(* IEC 61131-3 sources: Supremica/examples/ilprograms, 2 files *)

(* ---- ballProcess.il ---- *)
JAVA_BLOCK OnDelayTimer
	VAR_IN_OUT
		tonIN : BOOL;
		tonPT : DINT;
		tonET : DINT;
		tonQ  : BOOL;
	END_VAR
END_JAVA_BLOCK
FUNCTION_BLOCK TON
	VAR_IN_OUT
		tonIN : BOOL;
		tonPT : DINT;
		tonET : DINT;
		tonQ  : BOOL;
	END_VAR
	VAR
		odt : OnDelayTimer;
	END_VAR
	LD  tonIN
	ST  odt.tonIN
	LD  tonPT
	ST  odt.tonPT
	CAL odt
	LD  odt.tonET
	ST  tonET
	LD  odt.tonQ
	ST  tonQ
END_FUNCTION_BLOCK
(* This file is automatically generated from Supremica *)
(* Supremica version: 200206130257 *)
(* This file was generated at: Jun 13, 2002 6:24:47 AM *)
PROGRAM AutomaticallyGeneratedProgram
	VAR (* Internal variables *)
		si_6 AT %IX6 : BOOL; (* LitenKula *)
		si_2 AT %IX2 : BOOL; (* KulaMatlyft *)
		si_22 AT %IX22 : BOOL; (* KulaFast *)
		si_24 AT %IX24 : BOOL; (* ManuellStart *)
		si_16 AT %IX16 : BOOL; (* PlockaVan2 *)
		si_0 AT %IX0 : BOOL; (* KulaPortvakt *)
		si_13 AT %IX13 : BOOL; (* PlockaVan1 *)
		si_23 AT %IX23 : BOOL; (* Autostart *)
		si_4 AT %IX4 : BOOL; (* KulaMatstation *)
		si_14 AT %IX14 : BOOL; (* HissVan2 *)
		si_11 AT %IX11 : BOOL; (* HissVan1 *)
		si_15 AT %IX15 : BOOL; (* KulaVan2 *)
		si_12 AT %IX12 : BOOL; (* KulaVan1 *)
		si_25 AT %IX25 : BOOL; (* NodStopp *)
		si_21 AT %IX21 : BOOL; (* ArmVan2 *)
		si_3 AT %IX3 : BOOL; (* MatlyftUppe *)
		si_7 AT %IX7 : BOOL; (* HissNere *)
		si_20 AT %IX20 : BOOL; (* ArmVan1 *)
		si_17 AT %IX17 : BOOL; (* ArmHemma *)
		si_26 AT %IX26 : BOOL; (* LarmKvittering *)
		si_1 AT %IX1 : BOOL; (* MatlyftNere *)
		si_5 AT %IX5 : BOOL; (* StorKula *)
		si_10 AT %IX10 : BOOL; (* KulaHiss *)
		so_11 AT %QX11 : BOOL; (* UtVan2 *)
		so_7 AT %QX7 : BOOL; (* UtVan1 *)
		so_12 AT %QX12 : BOOL; (* LyftVan2 *)
		so_0 AT %QX0 : BOOL; (* InPortvakt *)
		so_10 AT %QX10 : BOOL; (* LyftVan1 *)
		so_15 AT %QX15 : BOOL; (* VridArmHoger *)
		so_3 AT %QX3 : BOOL; (* UrMatning *)
		so_14 AT %QX14 : BOOL; (* UppArmVan2 *)
		so_2 AT %QX2 : BOOL; (* UppMatlyft *)
		so_16 AT %QX16 : BOOL; (* Sug *)
		so_13 AT %QX13 : BOOL; (* UppArmVan1 *)
		so_6 AT %QX6 : BOOL; (* UppHissVan2 *)
		so_5 AT %QX5 : BOOL; (* UppHissVan1 *)
		so_1 AT %QX1 : BOOL; (* UrPortvakt *)
		so_4 AT %QX4 : BOOL; (* Mat *)
	END_VAR

	VAR (* Internal variables *)
		e_0 : BOOL; (* arm.allocate_lower_buffer controllable *)
		e_1 : BOOL; (* arm.allocate_upper_buffer controllable *)
		e_2 : BOOL; (* arm.lower_lower_buffer controllable *)
		e_3 : BOOL; (* arm.lower_upper_buffer controllable *)
		e_4 : BOOL; (* arm.raise_lower_buffer controllable *)
		e_5 : BOOL; (* arm.raise_upper_buffer controllable *)
		e_6 : BOOL; (* arm.release_lower_buffer controllable *)
		e_7 : BOOL; (* arm.release_upper_buffer controllable *)
		e_8 : BOOL; (* button.automatic.pressed uncontrollable *)
		e_9 : BOOL; (* button.automatic.released uncontrollable *)
		e_10 : BOOL; (* button.manual.pressed uncontrollable *)
		e_11 : BOOL; (* button.manual.released uncontrollable *)
		e_12 : BOOL; (* em.ball_out_of_measure_station uncontrollable *)
		e_13 : BOOL; (* em.elevator.allocate_station controllable *)
		e_14 : BOOL; (* em.elevator.release_station controllable *)
		e_15 : BOOL; (* em.enter_ball controllable *)
		e_16 : BOOL; (* em.go_down controllable *)
		e_17 : BOOL; (* em.go_up controllable *)
		e_18 : BOOL; (* em.has_ball uncontrollable *)
		e_19 : BOOL; (* em.is_down uncontrollable *)
		e_20 : BOOL; (* em.is_up uncontrollable *)
		e_21 : BOOL; (* em.large_ball uncontrollable *)
		e_22 : BOOL; (* em.measure.allocate_station controllable *)
		e_23 : BOOL; (* em.measure.finished uncontrollable *)
		e_24 : BOOL; (* em.measure.go_in controllable *)
		e_25 : BOOL; (* em.measure.go_out controllable *)
		e_26 : BOOL; (* em.measure.has_ball uncontrollable *)
		e_27 : BOOL; (* em.measure.has_no_ball uncontrollable *)
		e_28 : BOOL; (* em.measure.release_station controllable *)
		e_29 : BOOL; (* em.measure.start controllable *)
		e_30 : BOOL; (* em.putter.allocate_station controllable *)
		e_31 : BOOL; (* em.putter.finished uncontrollable *)
		e_32 : BOOL; (* em.putter.go_in controllable *)
		e_33 : BOOL; (* em.putter.go_out controllable *)
		e_34 : BOOL; (* em.putter.is_in controllable *)
		e_35 : BOOL; (* em.putter.is_out controllable *)
		e_36 : BOOL; (* em.putter.release_station controllable *)
		e_37 : BOOL; (* em.putter.start controllable *)
		e_38 : BOOL; (* em.small_ball uncontrollable *)
		e_39 : BOOL; (* em.timer.before_ballcheck.start controllable *)
		e_40 : BOOL; (* em.timer.before_ballcheck.timeout uncontrollable *)
		e_41 : BOOL; (* em.timer.before_put.start controllable *)
		e_42 : BOOL; (* em.timer.before_put.timeout uncontrollable *)
		e_43 : BOOL; (* em.timer.before_up.start controllable *)
		e_44 : BOOL; (* em.timer.before_up.timeout uncontrollable *)
		e_45 : BOOL; (* em.timer.measure.start controllable *)
		e_46 : BOOL; (* em.timer.measure.timeout uncontrollable *)
		e_47 : BOOL; (* em.timer.putting.start controllable *)
		e_48 : BOOL; (* em.timer.putting.timeout uncontrollable *)
		e_49 : BOOL; (* es.allocate_lower_buffer controllable *)
		e_50 : BOOL; (* es.allocate_upper_buffer controllable *)
		e_51 : BOOL; (* es.ball_lower_level uncontrollable *)
		e_52 : BOOL; (* es.ball_upper_level uncontrollable *)
		e_53 : BOOL; (* es.deput_ball_lower controllable *)
		e_54 : BOOL; (* es.deput_ball_upper controllable *)
		e_55 : BOOL; (* es.enter_ball controllable *)
		e_56 : BOOL; (* es.go_down controllable *)
		e_57 : BOOL; (* es.got_ball controllable *)
		e_58 : BOOL; (* es.is_lower uncontrollable *)
		e_59 : BOOL; (* es.is_not_down controllable *)
		e_60 : BOOL; (* es.is_upper uncontrollable *)
		e_61 : BOOL; (* es.lower_putter.go_in controllable *)
		e_62 : BOOL; (* es.lower_putter.go_out controllable *)
		e_63 : BOOL; (* es.no_ball_lower_level uncontrollable *)
		e_64 : BOOL; (* es.no_ball_upper_level uncontrollable *)
		e_65 : BOOL; (* es.put_ball_lower controllable *)
		e_66 : BOOL; (* es.put_ball_upper controllable *)
		e_67 : BOOL; (* es.release_lower_buffer controllable *)
		e_68 : BOOL; (* es.release_upper_buffer controllable *)
		e_69 : BOOL; (* es.timer.before_ballcheck.start controllable *)
		e_70 : BOOL; (* es.timer.before_ballcheck.timeout uncontrollable *)
		e_71 : BOOL; (* es.timer.before_deput.start controllable *)
		e_72 : BOOL; (* es.timer.before_deput.timeout uncontrollable *)
		e_73 : BOOL; (* es.timer.before_up.start controllable *)
		e_74 : BOOL; (* es.timer.before_up.timeout uncontrollable *)
		e_75 : BOOL; (* es.up_lower controllable *)
		e_76 : BOOL; (* es.up_upper controllable *)
		e_77 : BOOL; (* es.upper_putter.go_in controllable *)
		e_78 : BOOL; (* es.upper_putter.go_out controllable *)
		e_79 : BOOL; (* gk.ball_out_of_gatekeeper uncontrollable *)
		e_80 : BOOL; (* gk.enter_ball controllable *)
		e_81 : BOOL; (* gk.has_ball uncontrollable *)
		e_82 : BOOL; (* gk.in.go_in controllable *)
		e_83 : BOOL; (* gk.in.go_out controllable *)
		e_84 : BOOL; (* gk.in.is_in controllable *)
		e_85 : BOOL; (* gk.in.is_out controllable *)
		e_86 : BOOL; (* gk.out.go_in controllable *)
		e_87 : BOOL; (* gk.out.go_out controllable *)
		e_88 : BOOL; (* gk.out.is_in controllable *)
		e_89 : BOOL; (* gk.out.is_out controllable *)
		e_90 : BOOL; (* gk.release_ball controllable *)
		e_91 : BOOL; (* is_large_ball controllable *)
		e_92 : BOOL; (* is_small_ball controllable *)
		e_93 : BOOL; (* mode.automatic controllable *)
		e_94 : BOOL; (* mode.manual controllable *)
		enabledEvent : BOOL; (* True if a event is enabled, false otherwise *)
		q_0_0 : BOOL; (* q_0 in Progress spec: Manual or automatic mode *)
		q_0_1 : BOOL; (* q_1 in Progress spec: Manual or automatic mode *)
		q_0_2 : BOOL; (* q_2 in Progress spec: Manual or automatic mode *)
		q_0_3 : BOOL; (* q_3 in Progress spec: Manual or automatic mode *)
		q_0_4 : BOOL; (* q_4 in Progress spec: Manual or automatic mode *)
		q_0_5 : BOOL; (* q_5 in Progress spec: Manual or automatic mode *)
		q_0_6 : BOOL; (* q_6 in Progress spec: Manual or automatic mode *)
		q_0_7 : BOOL; (* q_7 in Progress spec: Manual or automatic mode *)
		q_1_0 : BOOL; (* q_0 in Progress spec: Gatekeeper (gk) *)
		q_1_1 : BOOL; (* q_1 in Progress spec: Gatekeeper (gk) *)
		q_1_2 : BOOL; (* q_1_1 in Progress spec: Gatekeeper (gk) *)
		q_1_3 : BOOL; (* q_2 in Progress spec: Gatekeeper (gk) *)
		q_1_4 : BOOL; (* q_3 in Progress spec: Gatekeeper (gk) *)
		q_1_5 : BOOL; (* q_4 in Progress spec: Gatekeeper (gk) *)
		q_1_6 : BOOL; (* q_5 in Progress spec: Gatekeeper (gk) *)
		q_1_7 : BOOL; (* q_6 in Progress spec: Gatekeeper (gk) *)
		q_2_0 : BOOL; (* q_0 in Progress spec: Elevate and measure (em) *)
		q_2_1 : BOOL; (* q_0_1 in Progress spec: Elevate and measure (em) *)
		q_2_2 : BOOL; (* q_1 in Progress spec: Elevate and measure (em) *)
		q_2_3 : BOOL; (* q_11 in Progress spec: Elevate and measure (em) *)
		q_2_4 : BOOL; (* q_11_1 in Progress spec: Elevate and measure (em) *)
		q_2_5 : BOOL; (* q_12 in Progress spec: Elevate and measure (em) *)
		q_2_6 : BOOL; (* q_12_1 in Progress spec: Elevate and measure (em) *)
		q_2_7 : BOOL; (* q_13 in Progress spec: Elevate and measure (em) *)
		q_2_8 : BOOL; (* q_2 in Progress spec: Elevate and measure (em) *)
		q_2_9 : BOOL; (* q_3 in Progress spec: Elevate and measure (em) *)
		q_2_10 : BOOL; (* q_3_1 in Progress spec: Elevate and measure (em) *)
		q_2_11 : BOOL; (* q_4 in Progress spec: Elevate and measure (em) *)
		q_2_12 : BOOL; (* q_5 in Progress spec: Elevate and measure (em) *)
		q_2_13 : BOOL; (* q_5_1 in Progress spec: Elevate and measure (em) *)
		q_2_14 : BOOL; (* q_6 in Progress spec: Elevate and measure (em) *)
		q_2_15 : BOOL; (* q_7 in Progress spec: Elevate and measure (em) *)
		q_2_16 : BOOL; (* q_8 in Progress spec: Elevate and measure (em) *)
		q_2_17 : BOOL; (* q_9 in Progress spec: Elevate and measure (em) *)
		q_2_18 : BOOL; (* q_9_1 in Progress spec: Elevate and measure (em) *)
		q_3_0 : BOOL; (* q_0 in Progress spec: Measure station - measure *)
		q_3_1 : BOOL; (* q_0_1 in Progress spec: Measure station - measure *)
		q_3_2 : BOOL; (* q_0_2 in Progress spec: Measure station - measure *)
		q_3_3 : BOOL; (* q_1 in Progress spec: Measure station - measure *)
		q_3_4 : BOOL; (* q_2 in Progress spec: Measure station - measure *)
		q_3_5 : BOOL; (* q_3 in Progress spec: Measure station - measure *)
		q_3_6 : BOOL; (* q_4 in Progress spec: Measure station - measure *)
		q_3_7 : BOOL; (* q_5 in Progress spec: Measure station - measure *)
		q_3_8 : BOOL; (* q_6 in Progress spec: Measure station - measure *)
		q_4_0 : BOOL; (* q_0 in Progress spec: Measure station - putter *)
		q_4_1 : BOOL; (* q_1 in Progress spec: Measure station - putter *)
		q_4_2 : BOOL; (* q_2 in Progress spec: Measure station - putter *)
		q_4_3 : BOOL; (* q_4 in Progress spec: Measure station - putter *)
		q_4_4 : BOOL; (* q_4_1 in Progress spec: Measure station - putter *)
		q_4_5 : BOOL; (* q_4_2 in Progress spec: Measure station - putter *)
		q_4_6 : BOOL; (* q_5 in Progress spec: Measure station - putter *)
		q_4_7 : BOOL; (* q_6 in Progress spec: Measure station - putter *)
		q_5_0 : BOOL; (* q_0 in Progress spec: Elevate and sort (es) *)
		q_5_1 : BOOL; (* q_0_1 in Progress spec: Elevate and sort (es) *)
		q_5_2 : BOOL; (* q_1 in Progress spec: Elevate and sort (es) *)
		q_5_3 : BOOL; (* q_10_lower in Progress spec: Elevate and sort (es) *)
		q_5_4 : BOOL; (* q_10_upper in Progress spec: Elevate and sort (es) *)
		q_5_5 : BOOL; (* q_11_lower in Progress spec: Elevate and sort (es) *)
		q_5_6 : BOOL; (* q_11_lower_1 in Progress spec: Elevate and sort (es) *)
		q_5_7 : BOOL; (* q_11_upper in Progress spec: Elevate and sort (es) *)
		q_5_8 : BOOL; (* q_11_upper_1 in Progress spec: Elevate and sort (es) *)
		q_5_9 : BOOL; (* q_12 in Progress spec: Elevate and sort (es) *)
		q_5_10 : BOOL; (* q_2 in Progress spec: Elevate and sort (es) *)
		q_5_11 : BOOL; (* q_3 in Progress spec: Elevate and sort (es) *)
		q_5_12 : BOOL; (* q_4_lower in Progress spec: Elevate and sort (es) *)
		q_5_13 : BOOL; (* q_4_upper in Progress spec: Elevate and sort (es) *)
		q_5_14 : BOOL; (* q_5_lower in Progress spec: Elevate and sort (es) *)
		q_5_15 : BOOL; (* q_5_upper in Progress spec: Elevate and sort (es) *)
		q_5_16 : BOOL; (* q_6_lower in Progress spec: Elevate and sort (es) *)
		q_5_17 : BOOL; (* q_6_upper in Progress spec: Elevate and sort (es) *)
		q_5_18 : BOOL; (* q_7_lower in Progress spec: Elevate and sort (es) *)
		q_5_19 : BOOL; (* q_7_upper in Progress spec: Elevate and sort (es) *)
		q_5_20 : BOOL; (* q_8_lower in Progress spec: Elevate and sort (es) *)
		q_5_21 : BOOL; (* q_8_lower_1 in Progress spec: Elevate and sort (es) *)
		q_5_22 : BOOL; (* q_8_lower_2 in Progress spec: Elevate and sort (es) *)
		q_5_23 : BOOL; (* q_8_upper in Progress spec: Elevate and sort (es) *)
		q_5_24 : BOOL; (* q_8_upper_1 in Progress spec: Elevate and sort (es) *)
		q_5_25 : BOOL; (* q_8_upper_2 in Progress spec: Elevate and sort (es) *)
		q_5_26 : BOOL; (* q_9_lower in Progress spec: Elevate and sort (es) *)
		q_5_27 : BOOL; (* q_9_upper in Progress spec: Elevate and sort (es) *)
		q_6_0 : BOOL; (* q_0 in Interaction spec: GK and EM *)
		q_6_1 : BOOL; (* q_1 in Interaction spec: GK and EM *)
		q_6_2 : BOOL; (* q_1_0 in Interaction spec: GK and EM *)
		q_6_3 : BOOL; (* q_2 in Interaction spec: GK and EM *)
		q_6_4 : BOOL; (* q_3 in Interaction spec: GK and EM *)
		q_6_5 : BOOL; (* q_4 in Interaction spec: GK and EM *)
		q_6_6 : BOOL; (* q_5 in Interaction spec: GK and EM *)
		q_7_0 : BOOL; (* q_0 in Interaction spec: Measure station *)
		q_7_1 : BOOL; (* q_1 in Interaction spec: Measure station *)
		q_7_2 : BOOL; (* q_2 in Interaction spec: Measure station *)
		q_7_3 : BOOL; (* q_3 in Interaction spec: Measure station *)
		q_8_0 : BOOL; (* q_0 in Interaction spec: EM and ES *)
		q_8_1 : BOOL; (* q_1 in Interaction spec: EM and ES *)
		q_9_0 : BOOL; (* q_0 in Interaction spec: ES and lower buffer *)
		q_9_1 : BOOL; (* q_1 in Interaction spec: ES and lower buffer *)
		q_9_2 : BOOL; (* q_2 in Interaction spec: ES and lower buffer *)
		q_10_0 : BOOL; (* q_0 in Interaction spec: ES and upper buffer *)
		q_10_1 : BOOL; (* q_1 in Interaction spec: ES and upper buffer *)
		q_10_2 : BOOL; (* q_2 in Interaction spec: ES and upper buffer *)
		q_11_0 : BOOL; (* q_0 in Plant: Manual button *)
		q_11_1 : BOOL; (* q_1 in Plant: Manual button *)
		q_11_2 : BOOL; (* q_2 in Plant: Manual button *)
		q_12_0 : BOOL; (* q_0 in Plant: Automatic button *)
		q_12_1 : BOOL; (* q_1 in Plant: Automatic button *)
		q_12_2 : BOOL; (* q_2 in Plant: Automatic button *)
		q_13_0 : BOOL; (* in in Plant: Gatekeeper - In *)
		q_13_1 : BOOL; (* out in Plant: Gatekeeper - In *)
		q_14_0 : BOOL; (* in in Plant: Gatekeeper - Out *)
		q_14_1 : BOOL; (* out in Plant: Gatekeeper - Out *)
		q_15_0 : BOOL; (* down in Plant: Elevator - Measure *)
		q_15_1 : BOOL; (* up in Plant: Elevator - Measure *)
		q_16_0 : BOOL; (* in in Plant: Measure - Putter *)
		q_16_1 : BOOL; (* out in Plant: Measure - Putter *)
		q_17_0 : BOOL; (* dummy in Plant: Disable events *)
		q_18_0 : BOOL; (* q_0 in Extended Plant: GK and EM *)
		q_18_1 : BOOL; (* q_1 in Extended Plant: GK and EM *)
		q_19_0 : BOOL; (* q_0 in Variable: size of ball *)
		q_19_1 : BOOL; (* q_1 in Variable: size of ball *)
		q_19_2 : BOOL; (* q_2 in Variable: size of ball *)
		q_20_0 : BOOL; (* q_0 in Timer: em.timer.before_up *)
		q_20_1 : BOOL; (* q_1 in Timer: em.timer.before_up *)
		q_21_0 : BOOL; (* q_0 in Timer: em.timer.before_ballcheck *)
		q_21_1 : BOOL; (* q_1 in Timer: em.timer.before_ballcheck *)
		q_22_0 : BOOL; (* q_0 in Timer: em.timer.measure *)
		q_22_1 : BOOL; (* q_1 in Timer: em.timer.measure *)
		q_23_0 : BOOL; (* q_0 in Timer: em.timer.before_put *)
		q_23_1 : BOOL; (* q_1 in Timer: em.timer.before_put *)
		q_24_0 : BOOL; (* q_0 in Timer: em.timer.putting *)
		q_24_1 : BOOL; (* q_1 in Timer: em.timer.putting *)
		q_25_0 : BOOL; (* q_0 in Timer: es.timer.before_up *)
		q_25_1 : BOOL; (* q_1 in Timer: es.timer.before_up *)
		q_26_0 : BOOL; (* q_0 in Timer: es.timer.before_ballcheck *)
		q_26_1 : BOOL; (* q_1 in Timer: es.timer.before_ballcheck *)
		q_27_0 : BOOL; (* q_0 in Timer: es.timer.before_deput *)
		q_27_1 : BOOL; (* q_1 in Timer: es.timer.before_deput *)
		initialized : BOOL; (* Set the inital state the first scan cycle *)
		timer_0 : TON; (* em.timer.before_up *)
		timer_1 : TON; (* es.timer.before_ballcheck *)
		timer_2 : TON; (* em.timer.before_put *)
		timer_3 : TON; (* es.timer.before_up *)
		timer_4 : TON; (* em.timer.measure *)
		timer_5 : TON; (* em.timer.putting *)
		timer_6 : TON; (* es.timer.before_deput *)
		timer_7 : TON; (* em.timer.before_ballcheck *)
	END_VAR

	(* Set the initial state *)
	LD	initialized
	JMPC	after_initialization
	LD	DINT#1000
	ST	timer_0.tonPT
	LD	DINT#1000
	ST	timer_1.tonPT
	LD	DINT#1000
	ST	timer_2.tonPT
	LD	DINT#1000
	ST	timer_3.tonPT
	LD	DINT#1000
	ST	timer_4.tonPT
	LD	DINT#2000
	ST	timer_5.tonPT
	LD	DINT#2000
	ST	timer_6.tonPT
	LD	DINT#1000
	ST	timer_7.tonPT
	LD	TRUE
	S	q_0_0
	S	q_1_0
	S	q_2_0
	S	q_3_0
	S	q_4_0
	S	q_5_0
	S	q_6_0
	S	q_7_0
	S	q_8_0
	S	q_9_0
	S	q_10_0
	S	q_11_0
	S	q_12_0
	S	q_13_0
	S	q_14_0
	S	q_15_0
	S	q_16_0
	S	q_17_0
	S	q_18_0
	S	q_19_0
	S	q_20_0
	S	q_21_0
	S	q_22_0
	S	q_23_0
	S	q_24_0
	S	q_25_0
	S	q_26_0
	S	q_27_0
	S	initialized
after_initialization:
	LD	FALSE
	ST	enabledEvent
	(* Compute the enabled events *)
	(* Enable condition for event "arm.allocate_lower_buffer" *)
	LD	q_9_0
	AND(	FALSE
	)
	ST	e_0
	(* Enable condition for event "arm.allocate_upper_buffer" *)
	LD	q_10_0
	AND(	FALSE
	)
	ST	e_1
	(* Enable condition for event "arm.lower_lower_buffer" *)
	LD	q_9_1
	ST	e_2
	(* Enable condition for event "arm.lower_upper_buffer" *)
	LD	q_10_1
	ST	e_3
	(* Enable condition for event "arm.raise_lower_buffer" *)
	LD	q_9_1
	ST	e_4
	(* Enable condition for event "arm.raise_upper_buffer" *)
	LD	q_10_1
	ST	e_5
	(* Enable condition for event "arm.release_lower_buffer" *)
	LD	q_9_1
	ST	e_6
	(* Enable condition for event "arm.release_upper_buffer" *)
	LD	q_10_1
	ST	e_7
	(* Enable condition for event "button.automatic.pressed" *)
	LD	q_12_0
	AND(	FALSE
	)
	ST	e_8
	(* Enable condition for event "button.automatic.released" *)
	LD	q_12_2
	ST	e_9
	(* Enable condition for event "button.manual.pressed" *)
	LD	q_11_0
	ST	e_10
	(* Enable condition for event "button.manual.released" *)
	LD	q_11_2
	ST	e_11
	(* Enable condition for event "em.ball_out_of_measure_station" *)
	LD	q_2_3
	ST	e_12
	(* Enable condition for event "em.elevator.allocate_station" *)
	LD	q_2_10
	OR	 q_2_6
	AND(	q_7_0
	)
	ST	e_13
	(* Enable condition for event "em.elevator.release_station" *)
	LD	q_2_13
	OR	 q_2_7
	AND(	q_7_3
	)
	ST	e_14
	(* Enable condition for event "em.enter_ball" *)
	LD	q_2_0
	AND(	q_6_1
	)
	ST	e_15
	(* Enable condition for event "em.go_down" *)
	LD	q_2_5
	AND(	q_7_3
	)
	AND(	q_15_0
	OR	 q_15_1
	)
	ST	e_16
	(* Enable condition for event "em.go_up" *)
	LD	q_2_9
	AND(	q_7_3
	)
	AND(	q_15_1
	OR	 q_15_0
	)
	ST	e_17
	(* Enable condition for event "em.has_ball" *)
	LD	q_2_1
	AND(	q_6_4
	)
	AND(	q_18_1
	)
	ST	e_18
	(* Enable condition for event "em.is_down" *)
	LD	q_6_2
	AND(	q_15_0
	)
	ST	e_19
	(* Enable condition for event "em.is_up" *)
	LD	q_2_11
	AND(	q_6_6
	)
	AND(	q_15_1
	)
	ST	e_20
	(* Enable condition for event "em.large_ball" *)
	LD	q_3_5
	AND(	q_19_0
	OR	 q_19_2
	)
	ST	e_21
	(* Enable condition for event "em.measure.allocate_station" *)
	LD	q_3_1
	AND(	q_7_0
	)
	ST	e_22
	(* Enable condition for event "em.measure.finished" *)
	LD	q_2_18
	AND(	q_3_8
	)
	ST	e_23
	(* Enable condition for event "em.measure.go_in" *)
	LD	q_3_6
	AND(	q_7_1
	)
	ST	e_24
	(* Enable condition for event "em.measure.go_out" *)
	LD	q_3_2
	AND(	q_7_1
	)
	ST	e_25
	(* Enable condition for event "em.measure.has_ball" *)
	LD	q_2_15
	AND(	q_8_0
	)
	ST	e_26
	(* Enable condition for event "em.measure.has_no_ball" *)
	LD	q_2_15
	ST	e_27
	(* Enable condition for event "em.measure.release_station" *)
	LD	q_3_7
	AND(	q_7_1
	)
	ST	e_28
	(* Enable condition for event "em.measure.start" *)
	LD	q_2_16
	AND(	q_3_0
	)
	ST	e_29
	(* Enable condition for event "em.putter.allocate_station" *)
	LD	q_4_1
	AND(	q_7_0
	)
	ST	e_30
	(* Enable condition for event "em.putter.finished" *)
	LD	q_2_4
	AND(	q_4_7
	)
	ST	e_31
	(* Enable condition for event "em.putter.go_in" *)
	LD	q_4_3
	AND(	q_7_2
	)
	AND(	q_16_0
	OR	 q_16_1
	)
	ST	e_32
	(* Enable condition for event "em.putter.go_out" *)
	LD	q_4_2
	AND(	q_7_2
	)
	AND(	q_16_1
	OR	 q_16_0
	)
	ST	e_33
	(* Enable condition for event "em.putter.is_in" *)
	LD	q_16_0
	AND(	FALSE
	)
	ST	e_34
	(* Enable condition for event "em.putter.is_out" *)
	LD	q_16_1
	AND(	FALSE
	)
	ST	e_35
	(* Enable condition for event "em.putter.release_station" *)
	LD	q_4_6
	AND(	q_7_2
	)
	ST	e_36
	(* Enable condition for event "em.putter.start" *)
	LD	q_2_17
	AND(	q_4_0
	)
	ST	e_37
	(* Enable condition for event "em.small_ball" *)
	LD	q_3_5
	AND(	q_19_0
	OR	 q_19_1
	)
	ST	e_38
	(* Enable condition for event "em.timer.before_ballcheck.start" *)
	LD	q_2_12
	AND(	q_21_0
	OR	 q_21_1
	)
	ST	e_39
	(* Enable condition for event "em.timer.before_ballcheck.timeout" *)
	LD	q_2_14
	AND(	q_21_1
	)
	ST	e_40
	(* Enable condition for event "em.timer.before_put.start" *)
	LD	FALSE
	AND(	q_23_0
	OR	 q_23_1
	)
	ST	e_41
	(* Enable condition for event "em.timer.before_put.timeout" *)
	LD	FALSE
	AND(	q_23_1
	)
	ST	e_42
	(* Enable condition for event "em.timer.before_up.start" *)
	LD	q_2_2
	AND(	q_20_0
	OR	 q_20_1
	)
	ST	e_43
	(* Enable condition for event "em.timer.before_up.timeout" *)
	LD	q_2_8
	AND(	q_20_1
	)
	ST	e_44
	(* Enable condition for event "em.timer.measure.start" *)
	LD	q_3_3
	AND(	q_22_0
	OR	 q_22_1
	)
	ST	e_45
	(* Enable condition for event "em.timer.measure.timeout" *)
	LD	q_3_4
	AND(	q_22_1
	)
	ST	e_46
	(* Enable condition for event "em.timer.putting.start" *)
	LD	q_4_4
	AND(	q_24_0
	OR	 q_24_1
	)
	ST	e_47
	(* Enable condition for event "em.timer.putting.timeout" *)
	LD	q_4_5
	AND(	q_24_1
	)
	ST	e_48
	(* Enable condition for event "es.allocate_lower_buffer" *)
	LD	q_5_20
	AND(	q_9_0
	)
	ST	e_49
	(* Enable condition for event "es.allocate_upper_buffer" *)
	LD	q_5_23
	AND(	q_10_0
	)
	ST	e_50
	(* Enable condition for event "es.ball_lower_level" *)
	LD	q_5_21
	ST	e_51
	(* Enable condition for event "es.ball_upper_level" *)
	LD	q_5_24
	ST	e_52
	(* Enable condition for event "es.deput_ball_lower" *)
	LD	q_9_2
	ST	e_53
	(* Enable condition for event "es.deput_ball_upper" *)
	LD	q_10_2
	ST	e_54
	(* Enable condition for event "es.enter_ball" *)
	LD	q_5_0
	AND(	q_8_1
	)
	ST	e_55
	(* Enable condition for event "es.go_down" *)
	LD	q_5_9
	ST	e_56
	(* Enable condition for event "es.got_ball" *)
	LD	q_5_1
	ST	e_57
	(* Enable condition for event "es.is_lower" *)
	LD	q_5_14
	ST	e_58
	(* Enable condition for event "es.is_not_down" *)
	LD	FALSE
	ST	e_59
	(* Enable condition for event "es.is_upper" *)
	LD	q_5_15
	ST	e_60
	(* Enable condition for event "es.lower_putter.go_in" *)
	LD	q_5_5
	ST	e_61
	(* Enable condition for event "es.lower_putter.go_out" *)
	LD	q_5_22
	ST	e_62
	(* Enable condition for event "es.no_ball_lower_level" *)
	LD	q_5_21
	ST	e_63
	(* Enable condition for event "es.no_ball_upper_level" *)
	LD	q_5_24
	ST	e_64
	(* Enable condition for event "es.put_ball_lower" *)
	LD	q_9_2
	ST	e_65
	(* Enable condition for event "es.put_ball_upper" *)
	LD	q_10_2
	ST	e_66
	(* Enable condition for event "es.release_lower_buffer" *)
	LD	q_5_6
	AND(	q_9_2
	)
	ST	e_67
	(* Enable condition for event "es.release_upper_buffer" *)
	LD	q_5_8
	AND(	q_10_2
	)
	ST	e_68
	(* Enable condition for event "es.timer.before_ballcheck.start" *)
	LD	q_5_16
	OR	 q_5_17
	AND(	q_26_0
	OR	 q_26_1
	)
	ST	e_69
	(* Enable condition for event "es.timer.before_ballcheck.timeout" *)
	LD	q_5_18
	OR	 q_5_19
	AND(	q_26_1
	)
	ST	e_70
	(* Enable condition for event "es.timer.before_deput.start" *)
	LD	q_5_26
	OR	 q_5_27
	AND(	q_27_0
	OR	 q_27_1
	)
	ST	e_71
	(* Enable condition for event "es.timer.before_deput.timeout" *)
	LD	q_5_3
	OR	 q_5_4
	AND(	q_27_1
	)
	ST	e_72
	(* Enable condition for event "es.timer.before_up.start" *)
	LD	q_5_2
	AND(	q_25_0
	OR	 q_25_1
	)
	ST	e_73
	(* Enable condition for event "es.timer.before_up.timeout" *)
	LD	q_5_10
	AND(	q_25_1
	)
	ST	e_74
	(* Enable condition for event "es.up_lower" *)
	LD	q_5_12
	ST	e_75
	(* Enable condition for event "es.up_upper" *)
	LD	q_5_13
	ST	e_76
	(* Enable condition for event "es.upper_putter.go_in" *)
	LD	q_5_7
	ST	e_77
	(* Enable condition for event "es.upper_putter.go_out" *)
	LD	q_5_25
	ST	e_78
	(* Enable condition for event "gk.ball_out_of_gatekeeper" *)
	LD	q_1_6
	AND(	q_6_5
	)
	ST	e_79
	(* Enable condition for event "gk.enter_ball" *)
	LD	q_0_1
	OR	 q_0_2
	OR	 q_0_3
	OR	 q_0_4
	OR	 q_0_5
	OR	 q_0_6
	OR	 q_0_7
	AND(	q_1_0
	)
	ST	e_80
	(* Enable condition for event "gk.has_ball" *)
	LD	q_1_1
	AND(	q_6_0
	)
	ST	e_81
	(* Enable condition for event "gk.in.go_in" *)
	LD	q_1_3
	AND(	q_13_0
	OR	 q_13_1
	)
	ST	e_82
	(* Enable condition for event "gk.in.go_out" *)
	LD	q_1_2
	AND(	q_13_1
	OR	 q_13_0
	)
	ST	e_83
	(* Enable condition for event "gk.in.is_in" *)
	LD	q_13_0
	AND(	FALSE
	)
	ST	e_84
	(* Enable condition for event "gk.in.is_out" *)
	LD	q_13_1
	AND(	FALSE
	)
	ST	e_85
	(* Enable condition for event "gk.out.go_in" *)
	LD	q_1_7
	AND(	q_14_0
	OR	 q_14_1
	)
	ST	e_86
	(* Enable condition for event "gk.out.go_out" *)
	LD	q_1_5
	AND(	q_14_1
	OR	 q_14_0
	)
	AND(	q_18_0
	)
	ST	e_87
	(* Enable condition for event "gk.out.is_in" *)
	LD	q_14_0
	AND(	FALSE
	)
	ST	e_88
	(* Enable condition for event "gk.out.is_out" *)
	LD	q_14_1
	AND(	FALSE
	)
	ST	e_89
	(* Enable condition for event "gk.release_ball" *)
	LD	q_1_4
	AND(	q_6_3
	)
	ST	e_90
	(* Enable condition for event "is_large_ball" *)
	LD	q_5_11
	AND(	q_19_1
	OR	 q_19_0
	)
	ST	e_91
	(* Enable condition for event "is_small_ball" *)
	LD	q_5_11
	AND(	q_19_2
	OR	 q_19_0
	)
	ST	e_92
	(* Enable condition for event "mode.automatic" *)
	LD	q_0_0
	OR	 q_0_1
	OR	 q_0_2
	OR	 q_0_3
	OR	 q_0_4
	OR	 q_0_5
	OR	 q_0_6
	OR	 q_0_7
	AND(	q_12_1
	)
	ST	e_93
	(* Enable condition for event "mode.manual" *)
	LD	q_0_0
	OR	 q_0_1
	OR	 q_0_2
	OR	 q_0_3
	OR	 q_0_4
	OR	 q_0_5
	OR	 q_0_6
	OR	 q_0_7
	AND(	q_11_1
	)
	ST	e_94
	(* Check if the events are externally enabled *)
	(* Enable condition for event "arm.allocate_lower_buffer" *)
	JMP	check_e_0
after_check_e_0:
	(* Enable condition for event "arm.allocate_upper_buffer" *)
	JMP	check_e_1
after_check_e_1:
	(* Enable condition for event "arm.lower_lower_buffer" *)
	JMP	check_e_2
after_check_e_2:
	(* Enable condition for event "arm.lower_upper_buffer" *)
	JMP	check_e_3
after_check_e_3:
	(* Enable condition for event "arm.raise_lower_buffer" *)
	JMP	check_e_4
after_check_e_4:
	(* Enable condition for event "arm.raise_upper_buffer" *)
	JMP	check_e_5
after_check_e_5:
	(* Enable condition for event "arm.release_lower_buffer" *)
	JMP	check_e_6
after_check_e_6:
	(* Enable condition for event "arm.release_upper_buffer" *)
	JMP	check_e_7
after_check_e_7:
	(* Enable condition for event "button.automatic.pressed" *)
	JMP	check_e_8
after_check_e_8:
	(* Enable condition for event "button.automatic.released" *)
	JMP	check_e_9
after_check_e_9:
	(* Enable condition for event "button.manual.pressed" *)
	JMP	check_e_10
after_check_e_10:
	(* Enable condition for event "button.manual.released" *)
	JMP	check_e_11
after_check_e_11:
	(* Enable condition for event "em.ball_out_of_measure_station" *)
	JMP	check_e_12
after_check_e_12:
	(* Enable condition for event "em.elevator.allocate_station" *)
	JMP	check_e_13
after_check_e_13:
	(* Enable condition for event "em.elevator.release_station" *)
	JMP	check_e_14
after_check_e_14:
	(* Enable condition for event "em.enter_ball" *)
	JMP	check_e_15
after_check_e_15:
	(* Enable condition for event "em.go_down" *)
	JMP	check_e_16
after_check_e_16:
	(* Enable condition for event "em.go_up" *)
	JMP	check_e_17
after_check_e_17:
	(* Enable condition for event "em.has_ball" *)
	JMP	check_e_18
after_check_e_18:
	(* Enable condition for event "em.is_down" *)
	JMP	check_e_19
after_check_e_19:
	(* Enable condition for event "em.is_up" *)
	JMP	check_e_20
after_check_e_20:
	(* Enable condition for event "em.large_ball" *)
	JMP	check_e_21
after_check_e_21:
	(* Enable condition for event "em.measure.allocate_station" *)
	JMP	check_e_22
after_check_e_22:
	(* Enable condition for event "em.measure.finished" *)
	JMP	check_e_23
after_check_e_23:
	(* Enable condition for event "em.measure.go_in" *)
	JMP	check_e_24
after_check_e_24:
	(* Enable condition for event "em.measure.go_out" *)
	JMP	check_e_25
after_check_e_25:
	(* Enable condition for event "em.measure.has_ball" *)
	JMP	check_e_26
after_check_e_26:
	(* Enable condition for event "em.measure.has_no_ball" *)
	JMP	check_e_27
after_check_e_27:
	(* Enable condition for event "em.measure.release_station" *)
	JMP	check_e_28
after_check_e_28:
	(* Enable condition for event "em.measure.start" *)
	JMP	check_e_29
after_check_e_29:
	(* Enable condition for event "em.putter.allocate_station" *)
	JMP	check_e_30
after_check_e_30:
	(* Enable condition for event "em.putter.finished" *)
	JMP	check_e_31
after_check_e_31:
	(* Enable condition for event "em.putter.go_in" *)
	JMP	check_e_32
after_check_e_32:
	(* Enable condition for event "em.putter.go_out" *)
	JMP	check_e_33
after_check_e_33:
	(* Enable condition for event "em.putter.is_in" *)
	JMP	check_e_34
after_check_e_34:
	(* Enable condition for event "em.putter.is_out" *)
	JMP	check_e_35
after_check_e_35:
	(* Enable condition for event "em.putter.release_station" *)
	JMP	check_e_36
after_check_e_36:
	(* Enable condition for event "em.putter.start" *)
	JMP	check_e_37
after_check_e_37:
	(* Enable condition for event "em.small_ball" *)
	JMP	check_e_38
after_check_e_38:
	(* Enable condition for event "em.timer.before_ballcheck.start" *)
	JMP	check_e_39
after_check_e_39:
	(* Enable condition for event "em.timer.before_ballcheck.timeout" *)
	JMP	check_e_40
after_check_e_40:
	(* Enable condition for event "em.timer.before_put.start" *)
	JMP	check_e_41
after_check_e_41:
	(* Enable condition for event "em.timer.before_put.timeout" *)
	JMP	check_e_42
after_check_e_42:
	(* Enable condition for event "em.timer.before_up.start" *)
	JMP	check_e_43
after_check_e_43:
	(* Enable condition for event "em.timer.before_up.timeout" *)
	JMP	check_e_44
after_check_e_44:
	(* Enable condition for event "em.timer.measure.start" *)
	JMP	check_e_45
after_check_e_45:
	(* Enable condition for event "em.timer.measure.timeout" *)
	JMP	check_e_46
after_check_e_46:
	(* Enable condition for event "em.timer.putting.start" *)
	JMP	check_e_47
after_check_e_47:
	(* Enable condition for event "em.timer.putting.timeout" *)
	JMP	check_e_48
after_check_e_48:
	(* Enable condition for event "es.allocate_lower_buffer" *)
	JMP	check_e_49
after_check_e_49:
	(* Enable condition for event "es.allocate_upper_buffer" *)
	JMP	check_e_50
after_check_e_50:
	(* Enable condition for event "es.ball_lower_level" *)
	JMP	check_e_51
after_check_e_51:
	(* Enable condition for event "es.ball_upper_level" *)
	JMP	check_e_52
after_check_e_52:
	(* Enable condition for event "es.deput_ball_lower" *)
	JMP	check_e_53
after_check_e_53:
	(* Enable condition for event "es.deput_ball_upper" *)
	JMP	check_e_54
after_check_e_54:
	(* Enable condition for event "es.enter_ball" *)
	JMP	check_e_55
after_check_e_55:
	(* Enable condition for event "es.go_down" *)
	JMP	check_e_56
after_check_e_56:
	(* Enable condition for event "es.got_ball" *)
	JMP	check_e_57
after_check_e_57:
	(* Enable condition for event "es.is_lower" *)
	JMP	check_e_58
after_check_e_58:
	(* Enable condition for event "es.is_not_down" *)
	JMP	check_e_59
after_check_e_59:
	(* Enable condition for event "es.is_upper" *)
	JMP	check_e_60
after_check_e_60:
	(* Enable condition for event "es.lower_putter.go_in" *)
	JMP	check_e_61
after_check_e_61:
	(* Enable condition for event "es.lower_putter.go_out" *)
	JMP	check_e_62
after_check_e_62:
	(* Enable condition for event "es.no_ball_lower_level" *)
	JMP	check_e_63
after_check_e_63:
	(* Enable condition for event "es.no_ball_upper_level" *)
	JMP	check_e_64
after_check_e_64:
	(* Enable condition for event "es.put_ball_lower" *)
	JMP	check_e_65
after_check_e_65:
	(* Enable condition for event "es.put_ball_upper" *)
	JMP	check_e_66
after_check_e_66:
	(* Enable condition for event "es.release_lower_buffer" *)
	JMP	check_e_67
after_check_e_67:
	(* Enable condition for event "es.release_upper_buffer" *)
	JMP	check_e_68
after_check_e_68:
	(* Enable condition for event "es.timer.before_ballcheck.start" *)
	JMP	check_e_69
after_check_e_69:
	(* Enable condition for event "es.timer.before_ballcheck.timeout" *)
	JMP	check_e_70
after_check_e_70:
	(* Enable condition for event "es.timer.before_deput.start" *)
	JMP	check_e_71
after_check_e_71:
	(* Enable condition for event "es.timer.before_deput.timeout" *)
	JMP	check_e_72
after_check_e_72:
	(* Enable condition for event "es.timer.before_up.start" *)
	JMP	check_e_73
after_check_e_73:
	(* Enable condition for event "es.timer.before_up.timeout" *)
	JMP	check_e_74
after_check_e_74:
	(* Enable condition for event "es.up_lower" *)
	JMP	check_e_75
after_check_e_75:
	(* Enable condition for event "es.up_upper" *)
	JMP	check_e_76
after_check_e_76:
	(* Enable condition for event "es.upper_putter.go_in" *)
	JMP	check_e_77
after_check_e_77:
	(* Enable condition for event "es.upper_putter.go_out" *)
	JMP	check_e_78
after_check_e_78:
	(* Enable condition for event "gk.ball_out_of_gatekeeper" *)
	JMP	check_e_79
after_check_e_79:
	(* Enable condition for event "gk.enter_ball" *)
	JMP	check_e_80
after_check_e_80:
	(* Enable condition for event "gk.has_ball" *)
	JMP	check_e_81
after_check_e_81:
	(* Enable condition for event "gk.in.go_in" *)
	JMP	check_e_82
after_check_e_82:
	(* Enable condition for event "gk.in.go_out" *)
	JMP	check_e_83
after_check_e_83:
	(* Enable condition for event "gk.in.is_in" *)
	JMP	check_e_84
after_check_e_84:
	(* Enable condition for event "gk.in.is_out" *)
	JMP	check_e_85
after_check_e_85:
	(* Enable condition for event "gk.out.go_in" *)
	JMP	check_e_86
after_check_e_86:
	(* Enable condition for event "gk.out.go_out" *)
	JMP	check_e_87
after_check_e_87:
	(* Enable condition for event "gk.out.is_in" *)
	JMP	check_e_88
after_check_e_88:
	(* Enable condition for event "gk.out.is_out" *)
	JMP	check_e_89
after_check_e_89:
	(* Enable condition for event "gk.release_ball" *)
	JMP	check_e_90
after_check_e_90:
	(* Enable condition for event "is_large_ball" *)
	JMP	check_e_91
after_check_e_91:
	(* Enable condition for event "is_small_ball" *)
	JMP	check_e_92
after_check_e_92:
	(* Enable condition for event "mode.automatic" *)
	JMP	check_e_93
after_check_e_93:
	(* Enable condition for event "mode.manual" *)
	JMP	check_e_94
after_check_e_94:
	(* Check if the events are enabled by timers *)
	(* Condition for timer em.timer.before_up *)
	(* Timeout event is "em.timer.before_up.timeout" *)
	LD	e_44
	JMPCN	after_check_timer_0
	CAL	timer_0
	LD	timer_0.tonQ
	JMPC	after_check_timer_0
	LD	FALSE
	ST	e_44
after_check_timer_0:
	(* Condition for timer es.timer.before_ballcheck *)
	(* Timeout event is "es.timer.before_ballcheck.timeout" *)
	LD	e_70
	JMPCN	after_check_timer_1
	CAL	timer_1
	LD	timer_1.tonQ
	JMPC	after_check_timer_1
	LD	FALSE
	ST	e_70
after_check_timer_1:
	(* Condition for timer em.timer.before_put *)
	(* Timeout event is "em.timer.before_put.timeout" *)
	LD	e_42
	JMPCN	after_check_timer_2
	CAL	timer_2
	LD	timer_2.tonQ
	JMPC	after_check_timer_2
	LD	FALSE
	ST	e_42
after_check_timer_2:
	(* Condition for timer es.timer.before_up *)
	(* Timeout event is "es.timer.before_up.timeout" *)
	LD	e_74
	JMPCN	after_check_timer_3
	CAL	timer_3
	LD	timer_3.tonQ
	JMPC	after_check_timer_3
	LD	FALSE
	ST	e_74
after_check_timer_3:
	(* Condition for timer em.timer.measure *)
	(* Timeout event is "em.timer.measure.timeout" *)
	LD	e_46
	JMPCN	after_check_timer_4
	CAL	timer_4
	LD	timer_4.tonQ
	JMPC	after_check_timer_4
	LD	FALSE
	ST	e_46
after_check_timer_4:
	(* Condition for timer em.timer.putting *)
	(* Timeout event is "em.timer.putting.timeout" *)
	LD	e_48
	JMPCN	after_check_timer_5
	CAL	timer_5
	LD	timer_5.tonQ
	JMPC	after_check_timer_5
	LD	FALSE
	ST	e_48
after_check_timer_5:
	(* Condition for timer es.timer.before_deput *)
	(* Timeout event is "es.timer.before_deput.timeout" *)
	LD	e_72
	JMPCN	after_check_timer_6
	CAL	timer_6
	LD	timer_6.tonQ
	JMPC	after_check_timer_6
	LD	FALSE
	ST	e_72
after_check_timer_6:
	(* Condition for timer em.timer.before_ballcheck *)
	(* Timeout event is "em.timer.before_ballcheck.timeout" *)
	LD	e_40
	JMPCN	after_check_timer_7
	CAL	timer_7
	LD	timer_7.tonQ
	JMPC	after_check_timer_7
	LD	FALSE
	ST	e_40
after_check_timer_7:
	(* Make sure only one event is enabled *)
	(* Priority is given to uncontrollable events *)
	(* Enable condition for event "button.automatic.pressed" *)
	LD	e_8
	ANDN	enabledEvent
	ST	e_8
	OR	enabledEvent
	ST	enabledEvent
	(* Enable condition for event "button.automatic.released" *)
	LD	e_9
	ANDN	enabledEvent
	ST	e_9
	OR	enabledEvent
	ST	enabledEvent
	(* Enable condition for event "button.manual.pressed" *)
	LD	e_10
	ANDN	enabledEvent
	ST	e_10
	OR	enabledEvent
	ST	enabledEvent
	(* Enable condition for event "button.manual.released" *)
	LD	e_11
	ANDN	enabledEvent
	ST	e_11
	OR	enabledEvent
	ST	enabledEvent
	(* Enable condition for event "em.ball_out_of_measure_station" *)
	LD	e_12
	ANDN	enabledEvent
	ST	e_12
	OR	enabledEvent
	ST	enabledEvent
	(* Enable condition for event "em.has_ball" *)
	LD	e_18
	ANDN	enabledEvent
	ST	e_18
	OR	enabledEvent
	ST	enabledEvent
	(* Enable condition for event "em.is_down" *)
	LD	e_19
	ANDN	enabledEvent
	ST	e_19
	OR	enabledEvent
	ST	enabledEvent
	(* Enable condition for event "em.is_up" *)
	LD	e_20
	ANDN	enabledEvent
	ST	e_20
	OR	enabledEvent
	ST	enabledEvent
	(* Enable condition for event "em.large_ball" *)
	LD	e_21
	ANDN	enabledEvent
	ST	e_21
	OR	enabledEvent
	ST	enabledEvent
	(* Enable condition for event "em.measure.finished" *)
	LD	e_23
	ANDN	enabledEvent
	ST	e_23
	OR	enabledEvent
	ST	enabledEvent
	(* Enable condition for event "em.measure.has_ball" *)
	LD	e_26
	ANDN	enabledEvent
	ST	e_26
	OR	enabledEvent
	ST	enabledEvent
	(* Enable condition for event "em.measure.has_no_ball" *)
	LD	e_27
	ANDN	enabledEvent
	ST	e_27
	OR	enabledEvent
	ST	enabledEvent
	(* Enable condition for event "em.putter.finished" *)
	LD	e_31
	ANDN	enabledEvent
	ST	e_31
	OR	enabledEvent
	ST	enabledEvent
	(* Enable condition for event "em.small_ball" *)
	LD	e_38
	ANDN	enabledEvent
	ST	e_38
	OR	enabledEvent
	ST	enabledEvent
	(* Enable condition for event "em.timer.before_ballcheck.timeout" *)
	LD	e_40
	ANDN	enabledEvent
	ST	e_40
	OR	enabledEvent
	ST	enabledEvent
	(* Enable condition for event "em.timer.before_put.timeout" *)
	LD	e_42
	ANDN	enabledEvent
	ST	e_42
	OR	enabledEvent
	ST	enabledEvent
	(* Enable condition for event "em.timer.before_up.timeout" *)
	LD	e_44
	ANDN	enabledEvent
	ST	e_44
	OR	enabledEvent
	ST	enabledEvent
	(* Enable condition for event "em.timer.measure.timeout" *)
	LD	e_46
	ANDN	enabledEvent
	ST	e_46
	OR	enabledEvent
	ST	enabledEvent
	(* Enable condition for event "em.timer.putting.timeout" *)
	LD	e_48
	ANDN	enabledEvent
	ST	e_48
	OR	enabledEvent
	ST	enabledEvent
	(* Enable condition for event "es.ball_lower_level" *)
	LD	e_51
	ANDN	enabledEvent
	ST	e_51
	OR	enabledEvent
	ST	enabledEvent
	(* Enable condition for event "es.ball_upper_level" *)
	LD	e_52
	ANDN	enabledEvent
	ST	e_52
	OR	enabledEvent
	ST	enabledEvent
	(* Enable condition for event "es.is_lower" *)
	LD	e_58
	ANDN	enabledEvent
	ST	e_58
	OR	enabledEvent
	ST	enabledEvent
	(* Enable condition for event "es.is_upper" *)
	LD	e_60
	ANDN	enabledEvent
	ST	e_60
	OR	enabledEvent
	ST	enabledEvent
	(* Enable condition for event "es.no_ball_lower_level" *)
	LD	e_63
	ANDN	enabledEvent
	ST	e_63
	OR	enabledEvent
	ST	enabledEvent
	(* Enable condition for event "es.no_ball_upper_level" *)
	LD	e_64
	ANDN	enabledEvent
	ST	e_64
	OR	enabledEvent
	ST	enabledEvent
	(* Enable condition for event "es.timer.before_ballcheck.timeout" *)
	LD	e_70
	ANDN	enabledEvent
	ST	e_70
	OR	enabledEvent
	ST	enabledEvent
	(* Enable condition for event "es.timer.before_deput.timeout" *)
	LD	e_72
	ANDN	enabledEvent
	ST	e_72
	OR	enabledEvent
	ST	enabledEvent
	(* Enable condition for event "es.timer.before_up.timeout" *)
	LD	e_74
	ANDN	enabledEvent
	ST	e_74
	OR	enabledEvent
	ST	enabledEvent
	(* Enable condition for event "gk.ball_out_of_gatekeeper" *)
	LD	e_79
	ANDN	enabledEvent
	ST	e_79
	OR	enabledEvent
	ST	enabledEvent
	(* Enable condition for event "gk.has_ball" *)
	LD	e_81
	ANDN	enabledEvent
	ST	e_81
	OR	enabledEvent
	ST	enabledEvent
	(* Enable condition for event "arm.allocate_lower_buffer" *)
	LD	e_0
	ANDN	enabledEvent
	ST	e_0
	OR	enabledEvent
	ST	enabledEvent
	(* Enable condition for event "arm.allocate_upper_buffer" *)
	LD	e_1
	ANDN	enabledEvent
	ST	e_1
	OR	enabledEvent
	ST	enabledEvent
	(* Enable condition for event "arm.lower_lower_buffer" *)
	LD	e_2
	ANDN	enabledEvent
	ST	e_2
	OR	enabledEvent
	ST	enabledEvent
	(* Enable condition for event "arm.lower_upper_buffer" *)
	LD	e_3
	ANDN	enabledEvent
	ST	e_3
	OR	enabledEvent
	ST	enabledEvent
	(* Enable condition for event "arm.raise_lower_buffer" *)
	LD	e_4
	ANDN	enabledEvent
	ST	e_4
	OR	enabledEvent
	ST	enabledEvent
	(* Enable condition for event "arm.raise_upper_buffer" *)
	LD	e_5
	ANDN	enabledEvent
	ST	e_5
	OR	enabledEvent
	ST	enabledEvent
	(* Enable condition for event "arm.release_lower_buffer" *)
	LD	e_6
	ANDN	enabledEvent
	ST	e_6
	OR	enabledEvent
	ST	enabledEvent
	(* Enable condition for event "arm.release_upper_buffer" *)
	LD	e_7
	ANDN	enabledEvent
	ST	e_7
	OR	enabledEvent
	ST	enabledEvent
	(* Enable condition for event "em.elevator.allocate_station" *)
	LD	e_13
	ANDN	enabledEvent
	ST	e_13
	OR	enabledEvent
	ST	enabledEvent
	(* Enable condition for event "em.elevator.release_station" *)
	LD	e_14
	ANDN	enabledEvent
	ST	e_14
	OR	enabledEvent
	ST	enabledEvent
	(* Enable condition for event "em.enter_ball" *)
	LD	e_15
	ANDN	enabledEvent
	ST	e_15
	OR	enabledEvent
	ST	enabledEvent
	(* Enable condition for event "em.go_down" *)
	LD	e_16
	ANDN	enabledEvent
	ST	e_16
	OR	enabledEvent
	ST	enabledEvent
	(* Enable condition for event "em.go_up" *)
	LD	e_17
	ANDN	enabledEvent
	ST	e_17
	OR	enabledEvent
	ST	enabledEvent
	(* Enable condition for event "em.measure.allocate_station" *)
	LD	e_22
	ANDN	enabledEvent
	ST	e_22
	OR	enabledEvent
	ST	enabledEvent
	(* Enable condition for event "em.measure.go_in" *)
	LD	e_24
	ANDN	enabledEvent
	ST	e_24
	OR	enabledEvent
	ST	enabledEvent
	(* Enable condition for event "em.measure.go_out" *)
	LD	e_25
	ANDN	enabledEvent
	ST	e_25
	OR	enabledEvent
	ST	enabledEvent
	(* Enable condition for event "em.measure.release_station" *)
	LD	e_28
	ANDN	enabledEvent
	ST	e_28
	OR	enabledEvent
	ST	enabledEvent
	(* Enable condition for event "em.measure.start" *)
	LD	e_29
	ANDN	enabledEvent
	ST	e_29
	OR	enabledEvent
	ST	enabledEvent
	(* Enable condition for event "em.putter.allocate_station" *)
	LD	e_30
	ANDN	enabledEvent
	ST	e_30
	OR	enabledEvent
	ST	enabledEvent
	(* Enable condition for event "em.putter.go_in" *)
	LD	e_32
	ANDN	enabledEvent
	ST	e_32
	OR	enabledEvent
	ST	enabledEvent
	(* Enable condition for event "em.putter.go_out" *)
	LD	e_33
	ANDN	enabledEvent
	ST	e_33
	OR	enabledEvent
	ST	enabledEvent
	(* Enable condition for event "em.putter.is_in" *)
	LD	e_34
	ANDN	enabledEvent
	ST	e_34
	OR	enabledEvent
	ST	enabledEvent
	(* Enable condition for event "em.putter.is_out" *)
	LD	e_35
	ANDN	enabledEvent
	ST	e_35
	OR	enabledEvent
	ST	enabledEvent
	(* Enable condition for event "em.putter.release_station" *)
	LD	e_36
	ANDN	enabledEvent
	ST	e_36
	OR	enabledEvent
	ST	enabledEvent
	(* Enable condition for event "em.putter.start" *)
	LD	e_37
	ANDN	enabledEvent
	ST	e_37
	OR	enabledEvent
	ST	enabledEvent
	(* Enable condition for event "em.timer.before_ballcheck.start" *)
	LD	e_39
	ANDN	enabledEvent
	ST	e_39
	OR	enabledEvent
	ST	enabledEvent
	(* Enable condition for event "em.timer.before_put.start" *)
	LD	e_41
	ANDN	enabledEvent
	ST	e_41
	OR	enabledEvent
	ST	enabledEvent
	(* Enable condition for event "em.timer.before_up.start" *)
	LD	e_43
	ANDN	enabledEvent
	ST	e_43
	OR	enabledEvent
	ST	enabledEvent
	(* Enable condition for event "em.timer.measure.start" *)
	LD	e_45
	ANDN	enabledEvent
	ST	e_45
	OR	enabledEvent
	ST	enabledEvent
	(* Enable condition for event "em.timer.putting.start" *)
	LD	e_47
	ANDN	enabledEvent
	ST	e_47
	OR	enabledEvent
	ST	enabledEvent
	(* Enable condition for event "es.allocate_lower_buffer" *)
	LD	e_49
	ANDN	enabledEvent
	ST	e_49
	OR	enabledEvent
	ST	enabledEvent
	(* Enable condition for event "es.allocate_upper_buffer" *)
	LD	e_50
	ANDN	enabledEvent
	ST	e_50
	OR	enabledEvent
	ST	enabledEvent
	(* Enable condition for event "es.deput_ball_lower" *)
	LD	e_53
	ANDN	enabledEvent
	ST	e_53
	OR	enabledEvent
	ST	enabledEvent
	(* Enable condition for event "es.deput_ball_upper" *)
	LD	e_54
	ANDN	enabledEvent
	ST	e_54
	OR	enabledEvent
	ST	enabledEvent
	(* Enable condition for event "es.enter_ball" *)
	LD	e_55
	ANDN	enabledEvent
	ST	e_55
	OR	enabledEvent
	ST	enabledEvent
	(* Enable condition for event "es.go_down" *)
	LD	e_56
	ANDN	enabledEvent
	ST	e_56
	OR	enabledEvent
	ST	enabledEvent
	(* Enable condition for event "es.got_ball" *)
	LD	e_57
	ANDN	enabledEvent
	ST	e_57
	OR	enabledEvent
	ST	enabledEvent
	(* Enable condition for event "es.is_not_down" *)
	LD	e_59
	ANDN	enabledEvent
	ST	e_59
	OR	enabledEvent
	ST	enabledEvent
	(* Enable condition for event "es.lower_putter.go_in" *)
	LD	e_61
	ANDN	enabledEvent
	ST	e_61
	OR	enabledEvent
	ST	enabledEvent
	(* Enable condition for event "es.lower_putter.go_out" *)
	LD	e_62
	ANDN	enabledEvent
	ST	e_62
	OR	enabledEvent
	ST	enabledEvent
	(* Enable condition for event "es.put_ball_lower" *)
	LD	e_65
	ANDN	enabledEvent
	ST	e_65
	OR	enabledEvent
	ST	enabledEvent
	(* Enable condition for event "es.put_ball_upper" *)
	LD	e_66
	ANDN	enabledEvent
	ST	e_66
	OR	enabledEvent
	ST	enabledEvent
	(* Enable condition for event "es.release_lower_buffer" *)
	LD	e_67
	ANDN	enabledEvent
	ST	e_67
	OR	enabledEvent
	ST	enabledEvent
	(* Enable condition for event "es.release_upper_buffer" *)
	LD	e_68
	ANDN	enabledEvent
	ST	e_68
	OR	enabledEvent
	ST	enabledEvent
	(* Enable condition for event "es.timer.before_ballcheck.start" *)
	LD	e_69
	ANDN	enabledEvent
	ST	e_69
	OR	enabledEvent
	ST	enabledEvent
	(* Enable condition for event "es.timer.before_deput.start" *)
	LD	e_71
	ANDN	enabledEvent
	ST	e_71
	OR	enabledEvent
	ST	enabledEvent
	(* Enable condition for event "es.timer.before_up.start" *)
	LD	e_73
	ANDN	enabledEvent
	ST	e_73
	OR	enabledEvent
	ST	enabledEvent
	(* Enable condition for event "es.up_lower" *)
	LD	e_75
	ANDN	enabledEvent
	ST	e_75
	OR	enabledEvent
	ST	enabledEvent
	(* Enable condition for event "es.up_upper" *)
	LD	e_76
	ANDN	enabledEvent
	ST	e_76
	OR	enabledEvent
	ST	enabledEvent
	(* Enable condition for event "es.upper_putter.go_in" *)
	LD	e_77
	ANDN	enabledEvent
	ST	e_77
	OR	enabledEvent
	ST	enabledEvent
	(* Enable condition for event "es.upper_putter.go_out" *)
	LD	e_78
	ANDN	enabledEvent
	ST	e_78
	OR	enabledEvent
	ST	enabledEvent
	(* Enable condition for event "gk.enter_ball" *)
	LD	e_80
	ANDN	enabledEvent
	ST	e_80
	OR	enabledEvent
	ST	enabledEvent
	(* Enable condition for event "gk.in.go_in" *)
	LD	e_82
	ANDN	enabledEvent
	ST	e_82
	OR	enabledEvent
	ST	enabledEvent
	(* Enable condition for event "gk.in.go_out" *)
	LD	e_83
	ANDN	enabledEvent
	ST	e_83
	OR	enabledEvent
	ST	enabledEvent
	(* Enable condition for event "gk.in.is_in" *)
	LD	e_84
	ANDN	enabledEvent
	ST	e_84
	OR	enabledEvent
	ST	enabledEvent
	(* Enable condition for event "gk.in.is_out" *)
	LD	e_85
	ANDN	enabledEvent
	ST	e_85
	OR	enabledEvent
	ST	enabledEvent
	(* Enable condition for event "gk.out.go_in" *)
	LD	e_86
	ANDN	enabledEvent
	ST	e_86
	OR	enabledEvent
	ST	enabledEvent
	(* Enable condition for event "gk.out.go_out" *)
	LD	e_87
	ANDN	enabledEvent
	ST	e_87
	OR	enabledEvent
	ST	enabledEvent
	(* Enable condition for event "gk.out.is_in" *)
	LD	e_88
	ANDN	enabledEvent
	ST	e_88
	OR	enabledEvent
	ST	enabledEvent
	(* Enable condition for event "gk.out.is_out" *)
	LD	e_89
	ANDN	enabledEvent
	ST	e_89
	OR	enabledEvent
	ST	enabledEvent
	(* Enable condition for event "gk.release_ball" *)
	LD	e_90
	ANDN	enabledEvent
	ST	e_90
	OR	enabledEvent
	ST	enabledEvent
	(* Enable condition for event "is_large_ball" *)
	LD	e_91
	ANDN	enabledEvent
	ST	e_91
	OR	enabledEvent
	ST	enabledEvent
	(* Enable condition for event "is_small_ball" *)
	LD	e_92
	ANDN	enabledEvent
	ST	e_92
	OR	enabledEvent
	ST	enabledEvent
	(* Enable condition for event "mode.automatic" *)
	LD	e_93
	ANDN	enabledEvent
	ST	e_93
	OR	enabledEvent
	ST	enabledEvent
	(* Enable condition for event "mode.manual" *)
	LD	e_94
	ANDN	enabledEvent
	ST	e_94
	OR	enabledEvent
	ST	enabledEvent
	(* Change state in the automata *)
	(* It is in general not safe to have more than one event set to true at this point *)
	(* Transition for event "arm.allocate_lower_buffer" *)
	LD	e_0
	JMPCN	trans_after_e_0
	JMP	do_e_0
after_do_e_0:
	(* Transitions in Interaction spec: ES and lower buffer *)
	LD	q_9_0
	JMPCN	trans_after_e_0_q_9_0
	S	q_9_1
	R	q_9_0
	JMP	trans_after_e_0_a_9
trans_after_e_0_q_9_0:
trans_after_e_0_a_9:
	(* Transitions in Plant: Disable events *)
trans_after_e_0_a_17:
trans_after_e_0:
	(* Transition for event "arm.allocate_upper_buffer" *)
	LD	e_1
	JMPCN	trans_after_e_1
	JMP	do_e_1
after_do_e_1:
	(* Transitions in Interaction spec: ES and upper buffer *)
	LD	q_10_0
	JMPCN	trans_after_e_1_q_10_0
	S	q_10_1
	R	q_10_0
	JMP	trans_after_e_1_a_10
trans_after_e_1_q_10_0:
trans_after_e_1_a_10:
	(* Transitions in Plant: Disable events *)
trans_after_e_1_a_17:
trans_after_e_1:
	(* Transition for event "arm.lower_lower_buffer" *)
	LD	e_2
	JMPCN	trans_after_e_2
	JMP	do_e_2
after_do_e_2:
	(* Transitions in Interaction spec: ES and lower buffer *)
	(* q_9_1  has e_2 as self loop, no transition *)
trans_after_e_2_q_9_1:
trans_after_e_2_a_9:
trans_after_e_2:
	(* Transition for event "arm.lower_upper_buffer" *)
	LD	e_3
	JMPCN	trans_after_e_3
	JMP	do_e_3
after_do_e_3:
	(* Transitions in Interaction spec: ES and upper buffer *)
	(* q_10_1  has e_3 as self loop, no transition *)
trans_after_e_3_q_10_1:
trans_after_e_3_a_10:
trans_after_e_3:
	(* Transition for event "arm.raise_lower_buffer" *)
	LD	e_4
	JMPCN	trans_after_e_4
	JMP	do_e_4
after_do_e_4:
	(* Transitions in Interaction spec: ES and lower buffer *)
	(* q_9_1  has e_4 as self loop, no transition *)
trans_after_e_4_q_9_1:
trans_after_e_4_a_9:
trans_after_e_4:
	(* Transition for event "arm.raise_upper_buffer" *)
	LD	e_5
	JMPCN	trans_after_e_5
	JMP	do_e_5
after_do_e_5:
	(* Transitions in Interaction spec: ES and upper buffer *)
	(* q_10_1  has e_5 as self loop, no transition *)
trans_after_e_5_q_10_1:
trans_after_e_5_a_10:
trans_after_e_5:
	(* Transition for event "arm.release_lower_buffer" *)
	LD	e_6
	JMPCN	trans_after_e_6
	JMP	do_e_6
after_do_e_6:
	(* Transitions in Interaction spec: ES and lower buffer *)
	LD	q_9_1
	JMPCN	trans_after_e_6_q_9_1
	S	q_9_0
	R	q_9_1
	JMP	trans_after_e_6_a_9
trans_after_e_6_q_9_1:
trans_after_e_6_a_9:
trans_after_e_6:
	(* Transition for event "arm.release_upper_buffer" *)
	LD	e_7
	JMPCN	trans_after_e_7
	JMP	do_e_7
after_do_e_7:
	(* Transitions in Interaction spec: ES and upper buffer *)
	LD	q_10_1
	JMPCN	trans_after_e_7_q_10_1
	S	q_10_0
	R	q_10_1
	JMP	trans_after_e_7_a_10
trans_after_e_7_q_10_1:
trans_after_e_7_a_10:
trans_after_e_7:
	(* Transition for event "button.automatic.pressed" *)
	LD	e_8
	JMPCN	trans_after_e_8
	JMP	do_e_8
after_do_e_8:
	(* Transitions in Plant: Automatic button *)
	LD	q_12_0
	JMPCN	trans_after_e_8_q_12_0
	S	q_12_1
	R	q_12_0
	JMP	trans_after_e_8_a_12
trans_after_e_8_q_12_0:
trans_after_e_8_a_12:
	(* Transitions in Plant: Disable events *)
trans_after_e_8_a_17:
trans_after_e_8:
	(* Transition for event "button.automatic.released" *)
	LD	e_9
	JMPCN	trans_after_e_9
	JMP	do_e_9
after_do_e_9:
	(* Transitions in Plant: Automatic button *)
	LD	q_12_2
	JMPCN	trans_after_e_9_q_12_2
	S	q_12_0
	R	q_12_2
	JMP	trans_after_e_9_a_12
trans_after_e_9_q_12_2:
trans_after_e_9_a_12:
trans_after_e_9:
	(* Transition for event "button.manual.pressed" *)
	LD	e_10
	JMPCN	trans_after_e_10
	JMP	do_e_10
after_do_e_10:
	(* Transitions in Plant: Manual button *)
	LD	q_11_0
	JMPCN	trans_after_e_10_q_11_0
	S	q_11_1
	R	q_11_0
	JMP	trans_after_e_10_a_11
trans_after_e_10_q_11_0:
trans_after_e_10_a_11:
trans_after_e_10:
	(* Transition for event "button.manual.released" *)
	LD	e_11
	JMPCN	trans_after_e_11
	JMP	do_e_11
after_do_e_11:
	(* Transitions in Plant: Manual button *)
	LD	q_11_2
	JMPCN	trans_after_e_11_q_11_2
	S	q_11_0
	R	q_11_2
	JMP	trans_after_e_11_a_11
trans_after_e_11_q_11_2:
trans_after_e_11_a_11:
trans_after_e_11:
	(* Transition for event "em.ball_out_of_measure_station" *)
	LD	e_12
	JMPCN	trans_after_e_12
	JMP	do_e_12
after_do_e_12:
	(* Transitions in Progress spec: Elevate and measure (em) *)
	LD	q_2_3
	JMPCN	trans_after_e_12_q_2_3
	S	q_2_6
	R	q_2_3
	JMP	trans_after_e_12_a_2
trans_after_e_12_q_2_3:
trans_after_e_12_a_2:
trans_after_e_12:
	(* Transition for event "em.elevator.allocate_station" *)
	LD	e_13
	JMPCN	trans_after_e_13
	JMP	do_e_13
after_do_e_13:
	(* Transitions in Progress spec: Elevate and measure (em) *)
	LD	q_2_10
	JMPCN	trans_after_e_13_q_2_10
	S	q_2_9
	R	q_2_10
	JMP	trans_after_e_13_a_2
trans_after_e_13_q_2_10:
	LD	q_2_6
	JMPCN	trans_after_e_13_q_2_6
	S	q_2_5
	R	q_2_6
	JMP	trans_after_e_13_a_2
trans_after_e_13_q_2_6:
trans_after_e_13_a_2:
	(* Transitions in Interaction spec: Measure station *)
	LD	q_7_0
	JMPCN	trans_after_e_13_q_7_0
	S	q_7_3
	R	q_7_0
	JMP	trans_after_e_13_a_7
trans_after_e_13_q_7_0:
trans_after_e_13_a_7:
trans_after_e_13:
	(* Transition for event "em.elevator.release_station" *)
	LD	e_14
	JMPCN	trans_after_e_14
	JMP	do_e_14
after_do_e_14:
	(* Transitions in Progress spec: Elevate and measure (em) *)
	LD	q_2_13
	JMPCN	trans_after_e_14_q_2_13
	S	q_2_12
	R	q_2_13
	JMP	trans_after_e_14_a_2
trans_after_e_14_q_2_13:
	LD	q_2_7
	JMPCN	trans_after_e_14_q_2_7
	S	q_2_0
	R	q_2_7
	JMP	trans_after_e_14_a_2
trans_after_e_14_q_2_7:
trans_after_e_14_a_2:
	(* Transitions in Interaction spec: Measure station *)
	LD	q_7_3
	JMPCN	trans_after_e_14_q_7_3
	S	q_7_0
	R	q_7_3
	JMP	trans_after_e_14_a_7
trans_after_e_14_q_7_3:
trans_after_e_14_a_7:
trans_after_e_14:
	(* Transition for event "em.enter_ball" *)
	LD	e_15
	JMPCN	trans_after_e_15
	JMP	do_e_15
after_do_e_15:
	(* Transitions in Progress spec: Elevate and measure (em) *)
	LD	q_2_0
	JMPCN	trans_after_e_15_q_2_0
	S	q_2_1
	R	q_2_0
	JMP	trans_after_e_15_a_2
trans_after_e_15_q_2_0:
trans_after_e_15_a_2:
	(* Transitions in Interaction spec: GK and EM *)
	LD	q_6_1
	JMPCN	trans_after_e_15_q_6_1
	S	q_6_3
	R	q_6_1
	JMP	trans_after_e_15_a_6
trans_after_e_15_q_6_1:
trans_after_e_15_a_6:
trans_after_e_15:
	(* Transition for event "em.go_down" *)
	LD	e_16
	JMPCN	trans_after_e_16
	JMP	do_e_16
after_do_e_16:
	(* Transitions in Progress spec: Elevate and measure (em) *)
	LD	q_2_5
	JMPCN	trans_after_e_16_q_2_5
	S	q_2_7
	R	q_2_5
	JMP	trans_after_e_16_a_2
trans_after_e_16_q_2_5:
trans_after_e_16_a_2:
	(* Transitions in Interaction spec: Measure station *)
	(* q_7_3  has e_16 as self loop, no transition *)
trans_after_e_16_q_7_3:
trans_after_e_16_a_7:
	(* Transitions in Plant: Elevator - Measure *)
	(* q_15_0  has e_16 as self loop, no transition *)
trans_after_e_16_q_15_0:
	LD	q_15_1
	JMPCN	trans_after_e_16_q_15_1
	S	q_15_0
	R	q_15_1
	JMP	trans_after_e_16_a_15
trans_after_e_16_q_15_1:
trans_after_e_16_a_15:
trans_after_e_16:
	(* Transition for event "em.go_up" *)
	LD	e_17
	JMPCN	trans_after_e_17
	JMP	do_e_17
after_do_e_17:
	(* Transitions in Progress spec: Elevate and measure (em) *)
	LD	q_2_9
	JMPCN	trans_after_e_17_q_2_9
	S	q_2_11
	R	q_2_9
	JMP	trans_after_e_17_a_2
trans_after_e_17_q_2_9:
trans_after_e_17_a_2:
	(* Transitions in Interaction spec: Measure station *)
	(* q_7_3  has e_17 as self loop, no transition *)
trans_after_e_17_q_7_3:
trans_after_e_17_a_7:
	(* Transitions in Plant: Elevator - Measure *)
	(* q_15_1  has e_17 as self loop, no transition *)
trans_after_e_17_q_15_1:
	LD	q_15_0
	JMPCN	trans_after_e_17_q_15_0
	S	q_15_1
	R	q_15_0
	JMP	trans_after_e_17_a_15
trans_after_e_17_q_15_0:
trans_after_e_17_a_15:
trans_after_e_17:
	(* Transition for event "em.has_ball" *)
	LD	e_18
	JMPCN	trans_after_e_18
	JMP	do_e_18
after_do_e_18:
	(* Transitions in Progress spec: Elevate and measure (em) *)
	LD	q_2_1
	JMPCN	trans_after_e_18_q_2_1
	S	q_2_2
	R	q_2_1
	JMP	trans_after_e_18_a_2
trans_after_e_18_q_2_1:
trans_after_e_18_a_2:
	(* Transitions in Interaction spec: GK and EM *)
	LD	q_6_4
	JMPCN	trans_after_e_18_q_6_4
	S	q_6_5
	R	q_6_4
	JMP	trans_after_e_18_a_6
trans_after_e_18_q_6_4:
trans_after_e_18_a_6:
	(* Transitions in Extended Plant: GK and EM *)
	LD	q_18_1
	JMPCN	trans_after_e_18_q_18_1
	S	q_18_0
	R	q_18_1
	JMP	trans_after_e_18_a_18
trans_after_e_18_q_18_1:
trans_after_e_18_a_18:
trans_after_e_18:
	(* Transition for event "em.is_down" *)
	LD	e_19
	JMPCN	trans_after_e_19
	JMP	do_e_19
after_do_e_19:
	(* Transitions in Interaction spec: GK and EM *)
	LD	q_6_2
	JMPCN	trans_after_e_19_q_6_2
	S	q_6_1
	R	q_6_2
	JMP	trans_after_e_19_a_6
trans_after_e_19_q_6_2:
trans_after_e_19_a_6:
	(* Transitions in Plant: Elevator - Measure *)
	(* q_15_0  has e_19 as self loop, no transition *)
trans_after_e_19_q_15_0:
trans_after_e_19_a_15:
trans_after_e_19:
	(* Transition for event "em.is_up" *)
	LD	e_20
	JMPCN	trans_after_e_20
	JMP	do_e_20
after_do_e_20:
	(* Transitions in Progress spec: Elevate and measure (em) *)
	LD	q_2_11
	JMPCN	trans_after_e_20_q_2_11
	S	q_2_13
	R	q_2_11
	JMP	trans_after_e_20_a_2
trans_after_e_20_q_2_11:
trans_after_e_20_a_2:
	(* Transitions in Interaction spec: GK and EM *)
	LD	q_6_6
	JMPCN	trans_after_e_20_q_6_6
	S	q_6_0
	R	q_6_6
	JMP	trans_after_e_20_a_6
trans_after_e_20_q_6_6:
trans_after_e_20_a_6:
	(* Transitions in Plant: Elevator - Measure *)
	(* q_15_1  has e_20 as self loop, no transition *)
trans_after_e_20_q_15_1:
trans_after_e_20_a_15:
trans_after_e_20:
	(* Transition for event "em.large_ball" *)
	LD	e_21
	JMPCN	trans_after_e_21
	JMP	do_e_21
after_do_e_21:
	(* Transitions in Progress spec: Measure station - measure *)
	LD	q_3_5
	JMPCN	trans_after_e_21_q_3_5
	S	q_3_6
	R	q_3_5
	JMP	trans_after_e_21_a_3
trans_after_e_21_q_3_5:
trans_after_e_21_a_3:
	(* Transitions in Variable: size of ball *)
	LD	q_19_0
	JMPCN	trans_after_e_21_q_19_0
	S	q_19_1
	R	q_19_0
	JMP	trans_after_e_21_a_19
trans_after_e_21_q_19_0:
	LD	q_19_2
	JMPCN	trans_after_e_21_q_19_2
	S	q_19_1
	R	q_19_2
	JMP	trans_after_e_21_a_19
trans_after_e_21_q_19_2:
trans_after_e_21_a_19:
trans_after_e_21:
	(* Transition for event "em.measure.allocate_station" *)
	LD	e_22
	JMPCN	trans_after_e_22
	JMP	do_e_22
after_do_e_22:
	(* Transitions in Progress spec: Measure station - measure *)
	LD	q_3_1
	JMPCN	trans_after_e_22_q_3_1
	S	q_3_2
	R	q_3_1
	JMP	trans_after_e_22_a_3
trans_after_e_22_q_3_1:
trans_after_e_22_a_3:
	(* Transitions in Interaction spec: Measure station *)
	LD	q_7_0
	JMPCN	trans_after_e_22_q_7_0
	S	q_7_1
	R	q_7_0
	JMP	trans_after_e_22_a_7
trans_after_e_22_q_7_0:
trans_after_e_22_a_7:
trans_after_e_22:
	(* Transition for event "em.measure.finished" *)
	LD	e_23
	JMPCN	trans_after_e_23
	JMP	do_e_23
after_do_e_23:
	(* Transitions in Progress spec: Elevate and measure (em) *)
	LD	q_2_18
	JMPCN	trans_after_e_23_q_2_18
	S	q_2_17
	R	q_2_18
	JMP	trans_after_e_23_a_2
trans_after_e_23_q_2_18:
trans_after_e_23_a_2:
	(* Transitions in Progress spec: Measure station - measure *)
	LD	q_3_8
	JMPCN	trans_after_e_23_q_3_8
	S	q_3_0
	R	q_3_8
	JMP	trans_after_e_23_a_3
trans_after_e_23_q_3_8:
trans_after_e_23_a_3:
trans_after_e_23:
	(* Transition for event "em.measure.go_in" *)
	LD	e_24
	JMPCN	trans_after_e_24
	JMP	do_e_24
after_do_e_24:
	(* Transitions in Progress spec: Measure station - measure *)
	LD	q_3_6
	JMPCN	trans_after_e_24_q_3_6
	S	q_3_7
	R	q_3_6
	JMP	trans_after_e_24_a_3
trans_after_e_24_q_3_6:
trans_after_e_24_a_3:
	(* Transitions in Interaction spec: Measure station *)
	(* q_7_1  has e_24 as self loop, no transition *)
trans_after_e_24_q_7_1:
trans_after_e_24_a_7:
trans_after_e_24:
	(* Transition for event "em.measure.go_out" *)
	LD	e_25
	JMPCN	trans_after_e_25
	JMP	do_e_25
after_do_e_25:
	(* Transitions in Progress spec: Measure station - measure *)
	LD	q_3_2
	JMPCN	trans_after_e_25_q_3_2
	S	q_3_3
	R	q_3_2
	JMP	trans_after_e_25_a_3
trans_after_e_25_q_3_2:
trans_after_e_25_a_3:
	(* Transitions in Interaction spec: Measure station *)
	(* q_7_1  has e_25 as self loop, no transition *)
trans_after_e_25_q_7_1:
trans_after_e_25_a_7:
trans_after_e_25:
	(* Transition for event "em.measure.has_ball" *)
	LD	e_26
	JMPCN	trans_after_e_26
	JMP	do_e_26
after_do_e_26:
	(* Transitions in Progress spec: Elevate and measure (em) *)
	LD	q_2_15
	JMPCN	trans_after_e_26_q_2_15
	S	q_2_16
	R	q_2_15
	JMP	trans_after_e_26_a_2
trans_after_e_26_q_2_15:
trans_after_e_26_a_2:
	(* Transitions in Interaction spec: EM and ES *)
	LD	q_8_0
	JMPCN	trans_after_e_26_q_8_0
	S	q_8_1
	R	q_8_0
	JMP	trans_after_e_26_a_8
trans_after_e_26_q_8_0:
trans_after_e_26_a_8:
trans_after_e_26:
	(* Transition for event "em.measure.has_no_ball" *)
	LD	e_27
	JMPCN	trans_after_e_27
	JMP	do_e_27
after_do_e_27:
	(* Transitions in Progress spec: Elevate and measure (em) *)
	LD	q_2_15
	JMPCN	trans_after_e_27_q_2_15
	S	q_2_5
	R	q_2_15
	JMP	trans_after_e_27_a_2
trans_after_e_27_q_2_15:
trans_after_e_27_a_2:
trans_after_e_27:
	(* Transition for event "em.measure.release_station" *)
	LD	e_28
	JMPCN	trans_after_e_28
	JMP	do_e_28
after_do_e_28:
	(* Transitions in Progress spec: Measure station - measure *)
	LD	q_3_7
	JMPCN	trans_after_e_28_q_3_7
	S	q_3_8
	R	q_3_7
	JMP	trans_after_e_28_a_3
trans_after_e_28_q_3_7:
trans_after_e_28_a_3:
	(* Transitions in Interaction spec: Measure station *)
	LD	q_7_1
	JMPCN	trans_after_e_28_q_7_1
	S	q_7_0
	R	q_7_1
	JMP	trans_after_e_28_a_7
trans_after_e_28_q_7_1:
trans_after_e_28_a_7:
trans_after_e_28:
	(* Transition for event "em.measure.start" *)
	LD	e_29
	JMPCN	trans_after_e_29
	JMP	do_e_29
after_do_e_29:
	(* Transitions in Progress spec: Elevate and measure (em) *)
	LD	q_2_16
	JMPCN	trans_after_e_29_q_2_16
	S	q_2_18
	R	q_2_16
	JMP	trans_after_e_29_a_2
trans_after_e_29_q_2_16:
trans_after_e_29_a_2:
	(* Transitions in Progress spec: Measure station - measure *)
	LD	q_3_0
	JMPCN	trans_after_e_29_q_3_0
	S	q_3_1
	R	q_3_0
	JMP	trans_after_e_29_a_3
trans_after_e_29_q_3_0:
trans_after_e_29_a_3:
trans_after_e_29:
	(* Transition for event "em.putter.allocate_station" *)
	LD	e_30
	JMPCN	trans_after_e_30
	JMP	do_e_30
after_do_e_30:
	(* Transitions in Progress spec: Measure station - putter *)
	LD	q_4_1
	JMPCN	trans_after_e_30_q_4_1
	S	q_4_2
	R	q_4_1
	JMP	trans_after_e_30_a_4
trans_after_e_30_q_4_1:
trans_after_e_30_a_4:
	(* Transitions in Interaction spec: Measure station *)
	LD	q_7_0
	JMPCN	trans_after_e_30_q_7_0
	S	q_7_2
	R	q_7_0
	JMP	trans_after_e_30_a_7
trans_after_e_30_q_7_0:
trans_after_e_30_a_7:
trans_after_e_30:
	(* Transition for event "em.putter.finished" *)
	LD	e_31
	JMPCN	trans_after_e_31
	JMP	do_e_31
after_do_e_31:
	(* Transitions in Progress spec: Elevate and measure (em) *)
	LD	q_2_4
	JMPCN	trans_after_e_31_q_2_4
	S	q_2_3
	R	q_2_4
	JMP	trans_after_e_31_a_2
trans_after_e_31_q_2_4:
trans_after_e_31_a_2:
	(* Transitions in Progress spec: Measure station - putter *)
	LD	q_4_7
	JMPCN	trans_after_e_31_q_4_7
	S	q_4_0
	R	q_4_7
	JMP	trans_after_e_31_a_4
trans_after_e_31_q_4_7:
trans_after_e_31_a_4:
trans_after_e_31:
	(* Transition for event "em.putter.go_in" *)
	LD	e_32
	JMPCN	trans_after_e_32
	JMP	do_e_32
after_do_e_32:
	(* Transitions in Progress spec: Measure station - putter *)
	LD	q_4_3
	JMPCN	trans_after_e_32_q_4_3
	S	q_4_6
	R	q_4_3
	JMP	trans_after_e_32_a_4
trans_after_e_32_q_4_3:
trans_after_e_32_a_4:
	(* Transitions in Interaction spec: Measure station *)
	(* q_7_2  has e_32 as self loop, no transition *)
trans_after_e_32_q_7_2:
trans_after_e_32_a_7:
	(* Transitions in Plant: Measure - Putter *)
	(* q_16_0  has e_32 as self loop, no transition *)
trans_after_e_32_q_16_0:
	LD	q_16_1
	JMPCN	trans_after_e_32_q_16_1
	S	q_16_0
	R	q_16_1
	JMP	trans_after_e_32_a_16
trans_after_e_32_q_16_1:
trans_after_e_32_a_16:
trans_after_e_32:
	(* Transition for event "em.putter.go_out" *)
	LD	e_33
	JMPCN	trans_after_e_33
	JMP	do_e_33
after_do_e_33:
	(* Transitions in Progress spec: Measure station - putter *)
	LD	q_4_2
	JMPCN	trans_after_e_33_q_4_2
	S	q_4_4
	R	q_4_2
	JMP	trans_after_e_33_a_4
trans_after_e_33_q_4_2:
trans_after_e_33_a_4:
	(* Transitions in Interaction spec: Measure station *)
	(* q_7_2  has e_33 as self loop, no transition *)
trans_after_e_33_q_7_2:
trans_after_e_33_a_7:
	(* Transitions in Plant: Measure - Putter *)
	(* q_16_1  has e_33 as self loop, no transition *)
trans_after_e_33_q_16_1:
	LD	q_16_0
	JMPCN	trans_after_e_33_q_16_0
	S	q_16_1
	R	q_16_0
	JMP	trans_after_e_33_a_16
trans_after_e_33_q_16_0:
trans_after_e_33_a_16:
trans_after_e_33:
	(* Transition for event "em.putter.is_in" *)
	LD	e_34
	JMPCN	trans_after_e_34
	JMP	do_e_34
after_do_e_34:
	(* Transitions in Plant: Measure - Putter *)
	(* q_16_0  has e_34 as self loop, no transition *)
trans_after_e_34_q_16_0:
trans_after_e_34_a_16:
	(* Transitions in Plant: Disable events *)
trans_after_e_34_a_17:
trans_after_e_34:
	(* Transition for event "em.putter.is_out" *)
	LD	e_35
	JMPCN	trans_after_e_35
	JMP	do_e_35
after_do_e_35:
	(* Transitions in Plant: Measure - Putter *)
	(* q_16_1  has e_35 as self loop, no transition *)
trans_after_e_35_q_16_1:
trans_after_e_35_a_16:
	(* Transitions in Plant: Disable events *)
trans_after_e_35_a_17:
trans_after_e_35:
	(* Transition for event "em.putter.release_station" *)
	LD	e_36
	JMPCN	trans_after_e_36
	JMP	do_e_36
after_do_e_36:
	(* Transitions in Progress spec: Measure station - putter *)
	LD	q_4_6
	JMPCN	trans_after_e_36_q_4_6
	S	q_4_7
	R	q_4_6
	JMP	trans_after_e_36_a_4
trans_after_e_36_q_4_6:
trans_after_e_36_a_4:
	(* Transitions in Interaction spec: Measure station *)
	LD	q_7_2
	JMPCN	trans_after_e_36_q_7_2
	S	q_7_0
	R	q_7_2
	JMP	trans_after_e_36_a_7
trans_after_e_36_q_7_2:
trans_after_e_36_a_7:
trans_after_e_36:
	(* Transition for event "em.putter.start" *)
	LD	e_37
	JMPCN	trans_after_e_37
	JMP	do_e_37
after_do_e_37:
	(* Transitions in Progress spec: Elevate and measure (em) *)
	LD	q_2_17
	JMPCN	trans_after_e_37_q_2_17
	S	q_2_4
	R	q_2_17
	JMP	trans_after_e_37_a_2
trans_after_e_37_q_2_17:
trans_after_e_37_a_2:
	(* Transitions in Progress spec: Measure station - putter *)
	LD	q_4_0
	JMPCN	trans_after_e_37_q_4_0
	S	q_4_1
	R	q_4_0
	JMP	trans_after_e_37_a_4
trans_after_e_37_q_4_0:
trans_after_e_37_a_4:
trans_after_e_37:
	(* Transition for event "em.small_ball" *)
	LD	e_38
	JMPCN	trans_after_e_38
	JMP	do_e_38
after_do_e_38:
	(* Transitions in Progress spec: Measure station - measure *)
	LD	q_3_5
	JMPCN	trans_after_e_38_q_3_5
	S	q_3_6
	R	q_3_5
	JMP	trans_after_e_38_a_3
trans_after_e_38_q_3_5:
trans_after_e_38_a_3:
	(* Transitions in Variable: size of ball *)
	LD	q_19_0
	JMPCN	trans_after_e_38_q_19_0
	S	q_19_2
	R	q_19_0
	JMP	trans_after_e_38_a_19
trans_after_e_38_q_19_0:
	LD	q_19_1
	JMPCN	trans_after_e_38_q_19_1
	S	q_19_2
	R	q_19_1
	JMP	trans_after_e_38_a_19
trans_after_e_38_q_19_1:
trans_after_e_38_a_19:
trans_after_e_38:
	(* Transition for event "em.timer.before_ballcheck.start" *)
	LD	e_39
	JMPCN	trans_after_e_39
	JMP	do_e_39
after_do_e_39:
	(* Transitions in Progress spec: Elevate and measure (em) *)
	LD	q_2_12
	JMPCN	trans_after_e_39_q_2_12
	S	q_2_14
	R	q_2_12
	JMP	trans_after_e_39_a_2
trans_after_e_39_q_2_12:
trans_after_e_39_a_2:
	(* Transitions in Timer: em.timer.before_ballcheck *)
	LD	q_21_0
	JMPCN	trans_after_e_39_q_21_0
	S	q_21_1
	R	q_21_0
	JMP	trans_after_e_39_a_21
trans_after_e_39_q_21_0:
	(* q_21_1  has e_39 as self loop, no transition *)
trans_after_e_39_q_21_1:
trans_after_e_39_a_21:
trans_after_e_39:
	(* Transition for event "em.timer.before_ballcheck.timeout" *)
	LD	e_40
	JMPCN	trans_after_e_40
	JMP	do_e_40
after_do_e_40:
	(* Transitions in Progress spec: Elevate and measure (em) *)
	LD	q_2_14
	JMPCN	trans_after_e_40_q_2_14
	S	q_2_15
	R	q_2_14
	JMP	trans_after_e_40_a_2
trans_after_e_40_q_2_14:
trans_after_e_40_a_2:
	(* Transitions in Timer: em.timer.before_ballcheck *)
	LD	q_21_1
	JMPCN	trans_after_e_40_q_21_1
	S	q_21_0
	R	q_21_1
	JMP	trans_after_e_40_a_21
trans_after_e_40_q_21_1:
trans_after_e_40_a_21:
trans_after_e_40:
	(* Transition for event "em.timer.before_put.start" *)
	LD	e_41
	JMPCN	trans_after_e_41
	JMP	do_e_41
after_do_e_41:
	(* Transitions in Progress spec: Elevate and measure (em) *)
trans_after_e_41_a_2:
	(* Transitions in Timer: em.timer.before_put *)
	LD	q_23_0
	JMPCN	trans_after_e_41_q_23_0
	S	q_23_1
	R	q_23_0
	JMP	trans_after_e_41_a_23
trans_after_e_41_q_23_0:
	(* q_23_1  has e_41 as self loop, no transition *)
trans_after_e_41_q_23_1:
trans_after_e_41_a_23:
trans_after_e_41:
	(* Transition for event "em.timer.before_put.timeout" *)
	LD	e_42
	JMPCN	trans_after_e_42
	JMP	do_e_42
after_do_e_42:
	(* Transitions in Progress spec: Elevate and measure (em) *)
trans_after_e_42_a_2:
	(* Transitions in Timer: em.timer.before_put *)
	LD	q_23_1
	JMPCN	trans_after_e_42_q_23_1
	S	q_23_0
	R	q_23_1
	JMP	trans_after_e_42_a_23
trans_after_e_42_q_23_1:
trans_after_e_42_a_23:
trans_after_e_42:
	(* Transition for event "em.timer.before_up.start" *)
	LD	e_43
	JMPCN	trans_after_e_43
	JMP	do_e_43
after_do_e_43:
	(* Transitions in Progress spec: Elevate and measure (em) *)
	LD	q_2_2
	JMPCN	trans_after_e_43_q_2_2
	S	q_2_8
	R	q_2_2
	JMP	trans_after_e_43_a_2
trans_after_e_43_q_2_2:
trans_after_e_43_a_2:
	(* Transitions in Timer: em.timer.before_up *)
	LD	q_20_0
	JMPCN	trans_after_e_43_q_20_0
	S	q_20_1
	R	q_20_0
	JMP	trans_after_e_43_a_20
trans_after_e_43_q_20_0:
	(* q_20_1  has e_43 as self loop, no transition *)
trans_after_e_43_q_20_1:
trans_after_e_43_a_20:
trans_after_e_43:
	(* Transition for event "em.timer.before_up.timeout" *)
	LD	e_44
	JMPCN	trans_after_e_44
	JMP	do_e_44
after_do_e_44:
	(* Transitions in Progress spec: Elevate and measure (em) *)
	LD	q_2_8
	JMPCN	trans_after_e_44_q_2_8
	S	q_2_10
	R	q_2_8
	JMP	trans_after_e_44_a_2
trans_after_e_44_q_2_8:
trans_after_e_44_a_2:
	(* Transitions in Timer: em.timer.before_up *)
	LD	q_20_1
	JMPCN	trans_after_e_44_q_20_1
	S	q_20_0
	R	q_20_1
	JMP	trans_after_e_44_a_20
trans_after_e_44_q_20_1:
trans_after_e_44_a_20:
trans_after_e_44:
	(* Transition for event "em.timer.measure.start" *)
	LD	e_45
	JMPCN	trans_after_e_45
	JMP	do_e_45
after_do_e_45:
	(* Transitions in Progress spec: Measure station - measure *)
	LD	q_3_3
	JMPCN	trans_after_e_45_q_3_3
	S	q_3_4
	R	q_3_3
	JMP	trans_after_e_45_a_3
trans_after_e_45_q_3_3:
trans_after_e_45_a_3:
	(* Transitions in Timer: em.timer.measure *)
	LD	q_22_0
	JMPCN	trans_after_e_45_q_22_0
	S	q_22_1
	R	q_22_0
	JMP	trans_after_e_45_a_22
trans_after_e_45_q_22_0:
	(* q_22_1  has e_45 as self loop, no transition *)
trans_after_e_45_q_22_1:
trans_after_e_45_a_22:
trans_after_e_45:
	(* Transition for event "em.timer.measure.timeout" *)
	LD	e_46
	JMPCN	trans_after_e_46
	JMP	do_e_46
after_do_e_46:
	(* Transitions in Progress spec: Measure station - measure *)
	LD	q_3_4
	JMPCN	trans_after_e_46_q_3_4
	S	q_3_5
	R	q_3_4
	JMP	trans_after_e_46_a_3
trans_after_e_46_q_3_4:
trans_after_e_46_a_3:
	(* Transitions in Timer: em.timer.measure *)
	LD	q_22_1
	JMPCN	trans_after_e_46_q_22_1
	S	q_22_0
	R	q_22_1
	JMP	trans_after_e_46_a_22
trans_after_e_46_q_22_1:
trans_after_e_46_a_22:
trans_after_e_46:
	(* Transition for event "em.timer.putting.start" *)
	LD	e_47
	JMPCN	trans_after_e_47
	JMP	do_e_47
after_do_e_47:
	(* Transitions in Progress spec: Measure station - putter *)
	LD	q_4_4
	JMPCN	trans_after_e_47_q_4_4
	S	q_4_5
	R	q_4_4
	JMP	trans_after_e_47_a_4
trans_after_e_47_q_4_4:
trans_after_e_47_a_4:
	(* Transitions in Timer: em.timer.putting *)
	LD	q_24_0
	JMPCN	trans_after_e_47_q_24_0
	S	q_24_1
	R	q_24_0
	JMP	trans_after_e_47_a_24
trans_after_e_47_q_24_0:
	(* q_24_1  has e_47 as self loop, no transition *)
trans_after_e_47_q_24_1:
trans_after_e_47_a_24:
trans_after_e_47:
	(* Transition for event "em.timer.putting.timeout" *)
	LD	e_48
	JMPCN	trans_after_e_48
	JMP	do_e_48
after_do_e_48:
	(* Transitions in Progress spec: Measure station - putter *)
	LD	q_4_5
	JMPCN	trans_after_e_48_q_4_5
	S	q_4_3
	R	q_4_5
	JMP	trans_after_e_48_a_4
trans_after_e_48_q_4_5:
trans_after_e_48_a_4:
	(* Transitions in Timer: em.timer.putting *)
	LD	q_24_1
	JMPCN	trans_after_e_48_q_24_1
	S	q_24_0
	R	q_24_1
	JMP	trans_after_e_48_a_24
trans_after_e_48_q_24_1:
trans_after_e_48_a_24:
trans_after_e_48:
	(* Transition for event "es.allocate_lower_buffer" *)
	LD	e_49
	JMPCN	trans_after_e_49
	JMP	do_e_49
after_do_e_49:
	(* Transitions in Progress spec: Elevate and sort (es) *)
	LD	q_5_20
	JMPCN	trans_after_e_49_q_5_20
	S	q_5_22
	R	q_5_20
	JMP	trans_after_e_49_a_5
trans_after_e_49_q_5_20:
trans_after_e_49_a_5:
	(* Transitions in Interaction spec: ES and lower buffer *)
	LD	q_9_0
	JMPCN	trans_after_e_49_q_9_0
	S	q_9_2
	R	q_9_0
	JMP	trans_after_e_49_a_9
trans_after_e_49_q_9_0:
trans_after_e_49_a_9:
trans_after_e_49:
	(* Transition for event "es.allocate_upper_buffer" *)
	LD	e_50
	JMPCN	trans_after_e_50
	JMP	do_e_50
after_do_e_50:
	(* Transitions in Progress spec: Elevate and sort (es) *)
	LD	q_5_23
	JMPCN	trans_after_e_50_q_5_23
	S	q_5_25
	R	q_5_23
	JMP	trans_after_e_50_a_5
trans_after_e_50_q_5_23:
trans_after_e_50_a_5:
	(* Transitions in Interaction spec: ES and upper buffer *)
	LD	q_10_0
	JMPCN	trans_after_e_50_q_10_0
	S	q_10_2
	R	q_10_0
	JMP	trans_after_e_50_a_10
trans_after_e_50_q_10_0:
trans_after_e_50_a_10:
trans_after_e_50:
	(* Transition for event "es.ball_lower_level" *)
	LD	e_51
	JMPCN	trans_after_e_51
	JMP	do_e_51
after_do_e_51:
	(* Transitions in Progress spec: Elevate and sort (es) *)
	LD	q_5_21
	JMPCN	trans_after_e_51_q_5_21
	S	q_5_20
	R	q_5_21
	JMP	trans_after_e_51_a_5
trans_after_e_51_q_5_21:
trans_after_e_51_a_5:
trans_after_e_51:
	(* Transition for event "es.ball_upper_level" *)
	LD	e_52
	JMPCN	trans_after_e_52
	JMP	do_e_52
after_do_e_52:
	(* Transitions in Progress spec: Elevate and sort (es) *)
	LD	q_5_24
	JMPCN	trans_after_e_52_q_5_24
	S	q_5_23
	R	q_5_24
	JMP	trans_after_e_52_a_5
trans_after_e_52_q_5_24:
trans_after_e_52_a_5:
trans_after_e_52:
	(* Transition for event "es.deput_ball_lower" *)
	LD	e_53
	JMPCN	trans_after_e_53
	JMP	do_e_53
after_do_e_53:
	(* Transitions in Interaction spec: ES and lower buffer *)
	(* q_9_2  has e_53 as self loop, no transition *)
trans_after_e_53_q_9_2:
trans_after_e_53_a_9:
trans_after_e_53:
	(* Transition for event "es.deput_ball_upper" *)
	LD	e_54
	JMPCN	trans_after_e_54
	JMP	do_e_54
after_do_e_54:
	(* Transitions in Interaction spec: ES and upper buffer *)
	(* q_10_2  has e_54 as self loop, no transition *)
trans_after_e_54_q_10_2:
trans_after_e_54_a_10:
trans_after_e_54:
	(* Transition for event "es.enter_ball" *)
	LD	e_55
	JMPCN	trans_after_e_55
	JMP	do_e_55
after_do_e_55:
	(* Transitions in Progress spec: Elevate and sort (es) *)
	LD	q_5_0
	JMPCN	trans_after_e_55_q_5_0
	S	q_5_1
	R	q_5_0
	JMP	trans_after_e_55_a_5
trans_after_e_55_q_5_0:
trans_after_e_55_a_5:
	(* Transitions in Interaction spec: EM and ES *)
	LD	q_8_1
	JMPCN	trans_after_e_55_q_8_1
	S	q_8_0
	R	q_8_1
	JMP	trans_after_e_55_a_8
trans_after_e_55_q_8_1:
trans_after_e_55_a_8:
trans_after_e_55:
	(* Transition for event "es.go_down" *)
	LD	e_56
	JMPCN	trans_after_e_56
	JMP	do_e_56
after_do_e_56:
	(* Transitions in Progress spec: Elevate and sort (es) *)
	LD	q_5_9
	JMPCN	trans_after_e_56_q_5_9
	S	q_5_0
	R	q_5_9
	JMP	trans_after_e_56_a_5
trans_after_e_56_q_5_9:
trans_after_e_56_a_5:
trans_after_e_56:
	(* Transition for event "es.got_ball" *)
	LD	e_57
	JMPCN	trans_after_e_57
	JMP	do_e_57
after_do_e_57:
	(* Transitions in Progress spec: Elevate and sort (es) *)
	LD	q_5_1
	JMPCN	trans_after_e_57_q_5_1
	S	q_5_2
	R	q_5_1
	JMP	trans_after_e_57_a_5
trans_after_e_57_q_5_1:
trans_after_e_57_a_5:
trans_after_e_57:
	(* Transition for event "es.is_lower" *)
	LD	e_58
	JMPCN	trans_after_e_58
	JMP	do_e_58
after_do_e_58:
	(* Transitions in Progress spec: Elevate and sort (es) *)
	LD	q_5_14
	JMPCN	trans_after_e_58_q_5_14
	S	q_5_16
	R	q_5_14
	JMP	trans_after_e_58_a_5
trans_after_e_58_q_5_14:
trans_after_e_58_a_5:
trans_after_e_58:
	(* Transition for event "es.is_not_down" *)
	LD	e_59
	JMPCN	trans_after_e_59
	JMP	do_e_59
after_do_e_59:
	(* Transitions in Progress spec: Elevate and sort (es) *)
trans_after_e_59_a_5:
trans_after_e_59:
	(* Transition for event "es.is_upper" *)
	LD	e_60
	JMPCN	trans_after_e_60
	JMP	do_e_60
after_do_e_60:
	(* Transitions in Progress spec: Elevate and sort (es) *)
	LD	q_5_15
	JMPCN	trans_after_e_60_q_5_15
	S	q_5_17
	R	q_5_15
	JMP	trans_after_e_60_a_5
trans_after_e_60_q_5_15:
trans_after_e_60_a_5:
trans_after_e_60:
	(* Transition for event "es.lower_putter.go_in" *)
	LD	e_61
	JMPCN	trans_after_e_61
	JMP	do_e_61
after_do_e_61:
	(* Transitions in Progress spec: Elevate and sort (es) *)
	LD	q_5_5
	JMPCN	trans_after_e_61_q_5_5
	S	q_5_6
	R	q_5_5
	JMP	trans_after_e_61_a_5
trans_after_e_61_q_5_5:
trans_after_e_61_a_5:
trans_after_e_61:
	(* Transition for event "es.lower_putter.go_out" *)
	LD	e_62
	JMPCN	trans_after_e_62
	JMP	do_e_62
after_do_e_62:
	(* Transitions in Progress spec: Elevate and sort (es) *)
	LD	q_5_22
	JMPCN	trans_after_e_62_q_5_22
	S	q_5_26
	R	q_5_22
	JMP	trans_after_e_62_a_5
trans_after_e_62_q_5_22:
trans_after_e_62_a_5:
trans_after_e_62:
	(* Transition for event "es.no_ball_lower_level" *)
	LD	e_63
	JMPCN	trans_after_e_63
	JMP	do_e_63
after_do_e_63:
	(* Transitions in Progress spec: Elevate and sort (es) *)
	LD	q_5_21
	JMPCN	trans_after_e_63_q_5_21
	S	q_5_9
	R	q_5_21
	JMP	trans_after_e_63_a_5
trans_after_e_63_q_5_21:
trans_after_e_63_a_5:
trans_after_e_63:
	(* Transition for event "es.no_ball_upper_level" *)
	LD	e_64
	JMPCN	trans_after_e_64
	JMP	do_e_64
after_do_e_64:
	(* Transitions in Progress spec: Elevate and sort (es) *)
	LD	q_5_24
	JMPCN	trans_after_e_64_q_5_24
	S	q_5_9
	R	q_5_24
	JMP	trans_after_e_64_a_5
trans_after_e_64_q_5_24:
trans_after_e_64_a_5:
trans_after_e_64:
	(* Transition for event "es.put_ball_lower" *)
	LD	e_65
	JMPCN	trans_after_e_65
	JMP	do_e_65
after_do_e_65:
	(* Transitions in Interaction spec: ES and lower buffer *)
	(* q_9_2  has e_65 as self loop, no transition *)
trans_after_e_65_q_9_2:
trans_after_e_65_a_9:
trans_after_e_65:
	(* Transition for event "es.put_ball_upper" *)
	LD	e_66
	JMPCN	trans_after_e_66
	JMP	do_e_66
after_do_e_66:
	(* Transitions in Interaction spec: ES and upper buffer *)
	(* q_10_2  has e_66 as self loop, no transition *)
trans_after_e_66_q_10_2:
trans_after_e_66_a_10:
trans_after_e_66:
	(* Transition for event "es.release_lower_buffer" *)
	LD	e_67
	JMPCN	trans_after_e_67
	JMP	do_e_67
after_do_e_67:
	(* Transitions in Progress spec: Elevate and sort (es) *)
	LD	q_5_6
	JMPCN	trans_after_e_67_q_5_6
	S	q_5_9
	R	q_5_6
	JMP	trans_after_e_67_a_5
trans_after_e_67_q_5_6:
trans_after_e_67_a_5:
	(* Transitions in Interaction spec: ES and lower buffer *)
	LD	q_9_2
	JMPCN	trans_after_e_67_q_9_2
	S	q_9_0
	R	q_9_2
	JMP	trans_after_e_67_a_9
trans_after_e_67_q_9_2:
trans_after_e_67_a_9:
trans_after_e_67:
	(* Transition for event "es.release_upper_buffer" *)
	LD	e_68
	JMPCN	trans_after_e_68
	JMP	do_e_68
after_do_e_68:
	(* Transitions in Progress spec: Elevate and sort (es) *)
	LD	q_5_8
	JMPCN	trans_after_e_68_q_5_8
	S	q_5_9
	R	q_5_8
	JMP	trans_after_e_68_a_5
trans_after_e_68_q_5_8:
trans_after_e_68_a_5:
	(* Transitions in Interaction spec: ES and upper buffer *)
	LD	q_10_2
	JMPCN	trans_after_e_68_q_10_2
	S	q_10_0
	R	q_10_2
	JMP	trans_after_e_68_a_10
trans_after_e_68_q_10_2:
trans_after_e_68_a_10:
trans_after_e_68:
	(* Transition for event "es.timer.before_ballcheck.start" *)
	LD	e_69
	JMPCN	trans_after_e_69
	JMP	do_e_69
after_do_e_69:
	(* Transitions in Progress spec: Elevate and sort (es) *)
	LD	q_5_16
	JMPCN	trans_after_e_69_q_5_16
	S	q_5_18
	R	q_5_16
	JMP	trans_after_e_69_a_5
trans_after_e_69_q_5_16:
	LD	q_5_17
	JMPCN	trans_after_e_69_q_5_17
	S	q_5_19
	R	q_5_17
	JMP	trans_after_e_69_a_5
trans_after_e_69_q_5_17:
trans_after_e_69_a_5:
	(* Transitions in Timer: es.timer.before_ballcheck *)
	LD	q_26_0
	JMPCN	trans_after_e_69_q_26_0
	S	q_26_1
	R	q_26_0
	JMP	trans_after_e_69_a_26
trans_after_e_69_q_26_0:
	(* q_26_1  has e_69 as self loop, no transition *)
trans_after_e_69_q_26_1:
trans_after_e_69_a_26:
trans_after_e_69:
	(* Transition for event "es.timer.before_ballcheck.timeout" *)
	LD	e_70
	JMPCN	trans_after_e_70
	JMP	do_e_70
after_do_e_70:
	(* Transitions in Progress spec: Elevate and sort (es) *)
	LD	q_5_18
	JMPCN	trans_after_e_70_q_5_18
	S	q_5_21
	R	q_5_18
	JMP	trans_after_e_70_a_5
trans_after_e_70_q_5_18:
	LD	q_5_19
	JMPCN	trans_after_e_70_q_5_19
	S	q_5_24
	R	q_5_19
	JMP	trans_after_e_70_a_5
trans_after_e_70_q_5_19:
trans_after_e_70_a_5:
	(* Transitions in Timer: es.timer.before_ballcheck *)
	LD	q_26_1
	JMPCN	trans_after_e_70_q_26_1
	S	q_26_0
	R	q_26_1
	JMP	trans_after_e_70_a_26
trans_after_e_70_q_26_1:
trans_after_e_70_a_26:
trans_after_e_70:
	(* Transition for event "es.timer.before_deput.start" *)
	LD	e_71
	JMPCN	trans_after_e_71
	JMP	do_e_71
after_do_e_71:
	(* Transitions in Progress spec: Elevate and sort (es) *)
	LD	q_5_26
	JMPCN	trans_after_e_71_q_5_26
	S	q_5_3
	R	q_5_26
	JMP	trans_after_e_71_a_5
trans_after_e_71_q_5_26:
	LD	q_5_27
	JMPCN	trans_after_e_71_q_5_27
	S	q_5_4
	R	q_5_27
	JMP	trans_after_e_71_a_5
trans_after_e_71_q_5_27:
trans_after_e_71_a_5:
	(* Transitions in Timer: es.timer.before_deput *)
	LD	q_27_0
	JMPCN	trans_after_e_71_q_27_0
	S	q_27_1
	R	q_27_0
	JMP	trans_after_e_71_a_27
trans_after_e_71_q_27_0:
	(* q_27_1  has e_71 as self loop, no transition *)
trans_after_e_71_q_27_1:
trans_after_e_71_a_27:
trans_after_e_71:
	(* Transition for event "es.timer.before_deput.timeout" *)
	LD	e_72
	JMPCN	trans_after_e_72
	JMP	do_e_72
after_do_e_72:
	(* Transitions in Progress spec: Elevate and sort (es) *)
	LD	q_5_3
	JMPCN	trans_after_e_72_q_5_3
	S	q_5_5
	R	q_5_3
	JMP	trans_after_e_72_a_5
trans_after_e_72_q_5_3:
	LD	q_5_4
	JMPCN	trans_after_e_72_q_5_4
	S	q_5_7
	R	q_5_4
	JMP	trans_after_e_72_a_5
trans_after_e_72_q_5_4:
trans_after_e_72_a_5:
	(* Transitions in Timer: es.timer.before_deput *)
	LD	q_27_1
	JMPCN	trans_after_e_72_q_27_1
	S	q_27_0
	R	q_27_1
	JMP	trans_after_e_72_a_27
trans_after_e_72_q_27_1:
trans_after_e_72_a_27:
trans_after_e_72:
	(* Transition for event "es.timer.before_up.start" *)
	LD	e_73
	JMPCN	trans_after_e_73
	JMP	do_e_73
after_do_e_73:
	(* Transitions in Progress spec: Elevate and sort (es) *)
	LD	q_5_2
	JMPCN	trans_after_e_73_q_5_2
	S	q_5_10
	R	q_5_2
	JMP	trans_after_e_73_a_5
trans_after_e_73_q_5_2:
trans_after_e_73_a_5:
	(* Transitions in Timer: es.timer.before_up *)
	LD	q_25_0
	JMPCN	trans_after_e_73_q_25_0
	S	q_25_1
	R	q_25_0
	JMP	trans_after_e_73_a_25
trans_after_e_73_q_25_0:
	(* q_25_1  has e_73 as self loop, no transition *)
trans_after_e_73_q_25_1:
trans_after_e_73_a_25:
trans_after_e_73:
	(* Transition for event "es.timer.before_up.timeout" *)
	LD	e_74
	JMPCN	trans_after_e_74
	JMP	do_e_74
after_do_e_74:
	(* Transitions in Progress spec: Elevate and sort (es) *)
	LD	q_5_10
	JMPCN	trans_after_e_74_q_5_10
	S	q_5_11
	R	q_5_10
	JMP	trans_after_e_74_a_5
trans_after_e_74_q_5_10:
trans_after_e_74_a_5:
	(* Transitions in Timer: es.timer.before_up *)
	LD	q_25_1
	JMPCN	trans_after_e_74_q_25_1
	S	q_25_0
	R	q_25_1
	JMP	trans_after_e_74_a_25
trans_after_e_74_q_25_1:
trans_after_e_74_a_25:
trans_after_e_74:
	(* Transition for event "es.up_lower" *)
	LD	e_75
	JMPCN	trans_after_e_75
	JMP	do_e_75
after_do_e_75:
	(* Transitions in Progress spec: Elevate and sort (es) *)
	LD	q_5_12
	JMPCN	trans_after_e_75_q_5_12
	S	q_5_14
	R	q_5_12
	JMP	trans_after_e_75_a_5
trans_after_e_75_q_5_12:
trans_after_e_75_a_5:
trans_after_e_75:
	(* Transition for event "es.up_upper" *)
	LD	e_76
	JMPCN	trans_after_e_76
	JMP	do_e_76
after_do_e_76:
	(* Transitions in Progress spec: Elevate and sort (es) *)
	LD	q_5_13
	JMPCN	trans_after_e_76_q_5_13
	S	q_5_15
	R	q_5_13
	JMP	trans_after_e_76_a_5
trans_after_e_76_q_5_13:
trans_after_e_76_a_5:
trans_after_e_76:
	(* Transition for event "es.upper_putter.go_in" *)
	LD	e_77
	JMPCN	trans_after_e_77
	JMP	do_e_77
after_do_e_77:
	(* Transitions in Progress spec: Elevate and sort (es) *)
	LD	q_5_7
	JMPCN	trans_after_e_77_q_5_7
	S	q_5_8
	R	q_5_7
	JMP	trans_after_e_77_a_5
trans_after_e_77_q_5_7:
trans_after_e_77_a_5:
trans_after_e_77:
	(* Transition for event "es.upper_putter.go_out" *)
	LD	e_78
	JMPCN	trans_after_e_78
	JMP	do_e_78
after_do_e_78:
	(* Transitions in Progress spec: Elevate and sort (es) *)
	LD	q_5_25
	JMPCN	trans_after_e_78_q_5_25
	S	q_5_27
	R	q_5_25
	JMP	trans_after_e_78_a_5
trans_after_e_78_q_5_25:
trans_after_e_78_a_5:
trans_after_e_78:
	(* Transition for event "gk.ball_out_of_gatekeeper" *)
	LD	e_79
	JMPCN	trans_after_e_79
	JMP	do_e_79
after_do_e_79:
	(* Transitions in Progress spec: Gatekeeper (gk) *)
	LD	q_1_6
	JMPCN	trans_after_e_79_q_1_6
	S	q_1_7
	R	q_1_6
	JMP	trans_after_e_79_a_1
trans_after_e_79_q_1_6:
trans_after_e_79_a_1:
	(* Transitions in Interaction spec: GK and EM *)
	LD	q_6_5
	JMPCN	trans_after_e_79_q_6_5
	S	q_6_6
	R	q_6_5
	JMP	trans_after_e_79_a_6
trans_after_e_79_q_6_5:
trans_after_e_79_a_6:
trans_after_e_79:
	(* Transition for event "gk.enter_ball" *)
	LD	e_80
	JMPCN	trans_after_e_80
	JMP	do_e_80
after_do_e_80:
	(* Transitions in Progress spec: Manual or automatic mode *)
	LD	q_0_1
	JMPCN	trans_after_e_80_q_0_1
	S	q_0_0
	R	q_0_1
	JMP	trans_after_e_80_a_0
trans_after_e_80_q_0_1:
	LD	q_0_2
	JMPCN	trans_after_e_80_q_0_2
	S	q_0_3
	R	q_0_2
	JMP	trans_after_e_80_a_0
trans_after_e_80_q_0_2:
	LD	q_0_3
	JMPCN	trans_after_e_80_q_0_3
	S	q_0_4
	R	q_0_3
	JMP	trans_after_e_80_a_0
trans_after_e_80_q_0_3:
	LD	q_0_4
	JMPCN	trans_after_e_80_q_0_4
	S	q_0_5
	R	q_0_4
	JMP	trans_after_e_80_a_0
trans_after_e_80_q_0_4:
	LD	q_0_5
	JMPCN	trans_after_e_80_q_0_5
	S	q_0_6
	R	q_0_5
	JMP	trans_after_e_80_a_0
trans_after_e_80_q_0_5:
	LD	q_0_6
	JMPCN	trans_after_e_80_q_0_6
	S	q_0_7
	R	q_0_6
	JMP	trans_after_e_80_a_0
trans_after_e_80_q_0_6:
	LD	q_0_7
	JMPCN	trans_after_e_80_q_0_7
	S	q_0_0
	R	q_0_7
	JMP	trans_after_e_80_a_0
trans_after_e_80_q_0_7:
trans_after_e_80_a_0:
	(* Transitions in Progress spec: Gatekeeper (gk) *)
	LD	q_1_0
	JMPCN	trans_after_e_80_q_1_0
	S	q_1_2
	R	q_1_0
	JMP	trans_after_e_80_a_1
trans_after_e_80_q_1_0:
trans_after_e_80_a_1:
trans_after_e_80:
	(* Transition for event "gk.has_ball" *)
	LD	e_81
	JMPCN	trans_after_e_81
	JMP	do_e_81
after_do_e_81:
	(* Transitions in Progress spec: Gatekeeper (gk) *)
	LD	q_1_1
	JMPCN	trans_after_e_81_q_1_1
	S	q_1_3
	R	q_1_1
	JMP	trans_after_e_81_a_1
trans_after_e_81_q_1_1:
trans_after_e_81_a_1:
	(* Transitions in Interaction spec: GK and EM *)
	LD	q_6_0
	JMPCN	trans_after_e_81_q_6_0
	S	q_6_2
	R	q_6_0
	JMP	trans_after_e_81_a_6
trans_after_e_81_q_6_0:
trans_after_e_81_a_6:
trans_after_e_81:
	(* Transition for event "gk.in.go_in" *)
	LD	e_82
	JMPCN	trans_after_e_82
	JMP	do_e_82
after_do_e_82:
	(* Transitions in Progress spec: Gatekeeper (gk) *)
	LD	q_1_3
	JMPCN	trans_after_e_82_q_1_3
	S	q_1_4
	R	q_1_3
	JMP	trans_after_e_82_a_1
trans_after_e_82_q_1_3:
trans_after_e_82_a_1:
	(* Transitions in Plant: Gatekeeper - In *)
	(* q_13_0  has e_82 as self loop, no transition *)
trans_after_e_82_q_13_0:
	LD	q_13_1
	JMPCN	trans_after_e_82_q_13_1
	S	q_13_0
	R	q_13_1
	JMP	trans_after_e_82_a_13
trans_after_e_82_q_13_1:
trans_after_e_82_a_13:
trans_after_e_82:
	(* Transition for event "gk.in.go_out" *)
	LD	e_83
	JMPCN	trans_after_e_83
	JMP	do_e_83
after_do_e_83:
	(* Transitions in Progress spec: Gatekeeper (gk) *)
	LD	q_1_2
	JMPCN	trans_after_e_83_q_1_2
	S	q_1_1
	R	q_1_2
	JMP	trans_after_e_83_a_1
trans_after_e_83_q_1_2:
trans_after_e_83_a_1:
	(* Transitions in Plant: Gatekeeper - In *)
	(* q_13_1  has e_83 as self loop, no transition *)
trans_after_e_83_q_13_1:
	LD	q_13_0
	JMPCN	trans_after_e_83_q_13_0
	S	q_13_1
	R	q_13_0
	JMP	trans_after_e_83_a_13
trans_after_e_83_q_13_0:
trans_after_e_83_a_13:
trans_after_e_83:
	(* Transition for event "gk.in.is_in" *)
	LD	e_84
	JMPCN	trans_after_e_84
	JMP	do_e_84
after_do_e_84:
	(* Transitions in Plant: Gatekeeper - In *)
	(* q_13_0  has e_84 as self loop, no transition *)
trans_after_e_84_q_13_0:
trans_after_e_84_a_13:
	(* Transitions in Plant: Disable events *)
trans_after_e_84_a_17:
trans_after_e_84:
	(* Transition for event "gk.in.is_out" *)
	LD	e_85
	JMPCN	trans_after_e_85
	JMP	do_e_85
after_do_e_85:
	(* Transitions in Plant: Gatekeeper - In *)
	(* q_13_1  has e_85 as self loop, no transition *)
trans_after_e_85_q_13_1:
trans_after_e_85_a_13:
	(* Transitions in Plant: Disable events *)
trans_after_e_85_a_17:
trans_after_e_85:
	(* Transition for event "gk.out.go_in" *)
	LD	e_86
	JMPCN	trans_after_e_86
	JMP	do_e_86
after_do_e_86:
	(* Transitions in Progress spec: Gatekeeper (gk) *)
	LD	q_1_7
	JMPCN	trans_after_e_86_q_1_7
	S	q_1_0
	R	q_1_7
	JMP	trans_after_e_86_a_1
trans_after_e_86_q_1_7:
trans_after_e_86_a_1:
	(* Transitions in Plant: Gatekeeper - Out *)
	(* q_14_0  has e_86 as self loop, no transition *)
trans_after_e_86_q_14_0:
	LD	q_14_1
	JMPCN	trans_after_e_86_q_14_1
	S	q_14_0
	R	q_14_1
	JMP	trans_after_e_86_a_14
trans_after_e_86_q_14_1:
trans_after_e_86_a_14:
trans_after_e_86:
	(* Transition for event "gk.out.go_out" *)
	LD	e_87
	JMPCN	trans_after_e_87
	JMP	do_e_87
after_do_e_87:
	(* Transitions in Progress spec: Gatekeeper (gk) *)
	LD	q_1_5
	JMPCN	trans_after_e_87_q_1_5
	S	q_1_6
	R	q_1_5
	JMP	trans_after_e_87_a_1
trans_after_e_87_q_1_5:
trans_after_e_87_a_1:
	(* Transitions in Plant: Gatekeeper - Out *)
	(* q_14_1  has e_87 as self loop, no transition *)
trans_after_e_87_q_14_1:
	LD	q_14_0
	JMPCN	trans_after_e_87_q_14_0
	S	q_14_1
	R	q_14_0
	JMP	trans_after_e_87_a_14
trans_after_e_87_q_14_0:
trans_after_e_87_a_14:
	(* Transitions in Extended Plant: GK and EM *)
	LD	q_18_0
	JMPCN	trans_after_e_87_q_18_0
	S	q_18_1
	R	q_18_0
	JMP	trans_after_e_87_a_18
trans_after_e_87_q_18_0:
trans_after_e_87_a_18:
trans_after_e_87:
	(* Transition for event "gk.out.is_in" *)
	LD	e_88
	JMPCN	trans_after_e_88
	JMP	do_e_88
after_do_e_88:
	(* Transitions in Plant: Gatekeeper - Out *)
	(* q_14_0  has e_88 as self loop, no transition *)
trans_after_e_88_q_14_0:
trans_after_e_88_a_14:
	(* Transitions in Plant: Disable events *)
trans_after_e_88_a_17:
trans_after_e_88:
	(* Transition for event "gk.out.is_out" *)
	LD	e_89
	JMPCN	trans_after_e_89
	JMP	do_e_89
after_do_e_89:
	(* Transitions in Plant: Gatekeeper - Out *)
	(* q_14_1  has e_89 as self loop, no transition *)
trans_after_e_89_q_14_1:
trans_after_e_89_a_14:
	(* Transitions in Plant: Disable events *)
trans_after_e_89_a_17:
trans_after_e_89:
	(* Transition for event "gk.release_ball" *)
	LD	e_90
	JMPCN	trans_after_e_90
	JMP	do_e_90
after_do_e_90:
	(* Transitions in Progress spec: Gatekeeper (gk) *)
	LD	q_1_4
	JMPCN	trans_after_e_90_q_1_4
	S	q_1_5
	R	q_1_4
	JMP	trans_after_e_90_a_1
trans_after_e_90_q_1_4:
trans_after_e_90_a_1:
	(* Transitions in Interaction spec: GK and EM *)
	LD	q_6_3
	JMPCN	trans_after_e_90_q_6_3
	S	q_6_4
	R	q_6_3
	JMP	trans_after_e_90_a_6
trans_after_e_90_q_6_3:
trans_after_e_90_a_6:
trans_after_e_90:
	(* Transition for event "is_large_ball" *)
	LD	e_91
	JMPCN	trans_after_e_91
	JMP	do_e_91
after_do_e_91:
	(* Transitions in Progress spec: Elevate and sort (es) *)
	LD	q_5_11
	JMPCN	trans_after_e_91_q_5_11
	S	q_5_13
	R	q_5_11
	JMP	trans_after_e_91_a_5
trans_after_e_91_q_5_11:
trans_after_e_91_a_5:
	(* Transitions in Variable: size of ball *)
	(* q_19_1  has e_91 as self loop, no transition *)
trans_after_e_91_q_19_1:
	(* q_19_0  has e_91 as self loop, no transition *)
trans_after_e_91_q_19_0:
trans_after_e_91_a_19:
trans_after_e_91:
	(* Transition for event "is_small_ball" *)
	LD	e_92
	JMPCN	trans_after_e_92
	JMP	do_e_92
after_do_e_92:
	(* Transitions in Progress spec: Elevate and sort (es) *)
	LD	q_5_11
	JMPCN	trans_after_e_92_q_5_11
	S	q_5_12
	R	q_5_11
	JMP	trans_after_e_92_a_5
trans_after_e_92_q_5_11:
trans_after_e_92_a_5:
	(* Transitions in Variable: size of ball *)
	(* q_19_2  has e_92 as self loop, no transition *)
trans_after_e_92_q_19_2:
	(* q_19_0  has e_92 as self loop, no transition *)
trans_after_e_92_q_19_0:
trans_after_e_92_a_19:
trans_after_e_92:
	(* Transition for event "mode.automatic" *)
	LD	e_93
	JMPCN	trans_after_e_93
	JMP	do_e_93
after_do_e_93:
	(* Transitions in Progress spec: Manual or automatic mode *)
	LD	q_0_0
	JMPCN	trans_after_e_93_q_0_0
	S	q_0_2
	R	q_0_0
	JMP	trans_after_e_93_a_0
trans_after_e_93_q_0_0:
	(* q_0_1  has e_93 as self loop, no transition *)
trans_after_e_93_q_0_1:
	(* q_0_2  has e_93 as self loop, no transition *)
trans_after_e_93_q_0_2:
	(* q_0_3  has e_93 as self loop, no transition *)
trans_after_e_93_q_0_3:
	(* q_0_4  has e_93 as self loop, no transition *)
trans_after_e_93_q_0_4:
	(* q_0_5  has e_93 as self loop, no transition *)
trans_after_e_93_q_0_5:
	(* q_0_6  has e_93 as self loop, no transition *)
trans_after_e_93_q_0_6:
	(* q_0_7  has e_93 as self loop, no transition *)
trans_after_e_93_q_0_7:
trans_after_e_93_a_0:
	(* Transitions in Plant: Automatic button *)
	LD	q_12_1
	JMPCN	trans_after_e_93_q_12_1
	S	q_12_2
	R	q_12_1
	JMP	trans_after_e_93_a_12
trans_after_e_93_q_12_1:
trans_after_e_93_a_12:
trans_after_e_93:
	(* Transition for event "mode.manual" *)
	LD	e_94
	JMPCN	trans_after_e_94
	JMP	do_e_94
after_do_e_94:
	(* Transitions in Progress spec: Manual or automatic mode *)
	LD	q_0_0
	JMPCN	trans_after_e_94_q_0_0
	S	q_0_1
	R	q_0_0
	JMP	trans_after_e_94_a_0
trans_after_e_94_q_0_0:
	(* q_0_1  has e_94 as self loop, no transition *)
trans_after_e_94_q_0_1:
	(* q_0_2  has e_94 as self loop, no transition *)
trans_after_e_94_q_0_2:
	(* q_0_3  has e_94 as self loop, no transition *)
trans_after_e_94_q_0_3:
	(* q_0_4  has e_94 as self loop, no transition *)
trans_after_e_94_q_0_4:
	(* q_0_5  has e_94 as self loop, no transition *)
trans_after_e_94_q_0_5:
	(* q_0_6  has e_94 as self loop, no transition *)
trans_after_e_94_q_0_6:
	(* q_0_7  has e_94 as self loop, no transition *)
trans_after_e_94_q_0_7:
trans_after_e_94_a_0:
	(* Transitions in Plant: Manual button *)
	LD	q_11_1
	JMPCN	trans_after_e_94_q_11_1
	S	q_11_2
	R	q_11_1
	JMP	trans_after_e_94_a_11
trans_after_e_94_q_11_1:
trans_after_e_94_a_11:
trans_after_e_94:
	(* Start timers *)
	(* Start timer em.timer.before_up *)
	(* Start event is "em.timer.before_up.start" *)
	LD	e_43
	JMPCN	after_start_timer_0
	LD	FALSE
	ST	timer_0.tonIN
	CAL	timer_0
	LD	TRUE
	ST	timer_0.tonIN
	CAL	timer_0
after_start_timer_0:
	(* Start timer es.timer.before_ballcheck *)
	(* Start event is "es.timer.before_ballcheck.start" *)
	LD	e_69
	JMPCN	after_start_timer_1
	LD	FALSE
	ST	timer_1.tonIN
	CAL	timer_1
	LD	TRUE
	ST	timer_1.tonIN
	CAL	timer_1
after_start_timer_1:
	(* Start timer em.timer.before_put *)
	(* Start event is "em.timer.before_put.start" *)
	LD	e_41
	JMPCN	after_start_timer_2
	LD	FALSE
	ST	timer_2.tonIN
	CAL	timer_2
	LD	TRUE
	ST	timer_2.tonIN
	CAL	timer_2
after_start_timer_2:
	(* Start timer es.timer.before_up *)
	(* Start event is "es.timer.before_up.start" *)
	LD	e_73
	JMPCN	after_start_timer_3
	LD	FALSE
	ST	timer_3.tonIN
	CAL	timer_3
	LD	TRUE
	ST	timer_3.tonIN
	CAL	timer_3
after_start_timer_3:
	(* Start timer em.timer.measure *)
	(* Start event is "em.timer.measure.start" *)
	LD	e_45
	JMPCN	after_start_timer_4
	LD	FALSE
	ST	timer_4.tonIN
	CAL	timer_4
	LD	TRUE
	ST	timer_4.tonIN
	CAL	timer_4
after_start_timer_4:
	(* Start timer em.timer.putting *)
	(* Start event is "em.timer.putting.start" *)
	LD	e_47
	JMPCN	after_start_timer_5
	LD	FALSE
	ST	timer_5.tonIN
	CAL	timer_5
	LD	TRUE
	ST	timer_5.tonIN
	CAL	timer_5
after_start_timer_5:
	(* Start timer es.timer.before_deput *)
	(* Start event is "es.timer.before_deput.start" *)
	LD	e_71
	JMPCN	after_start_timer_6
	LD	FALSE
	ST	timer_6.tonIN
	CAL	timer_6
	LD	TRUE
	ST	timer_6.tonIN
	CAL	timer_6
after_start_timer_6:
	(* Start timer em.timer.before_ballcheck *)
	(* Start event is "em.timer.before_ballcheck.start" *)
	LD	e_39
	JMPCN	after_start_timer_7
	LD	FALSE
	ST	timer_7.tonIN
	CAL	timer_7
	LD	TRUE
	ST	timer_7.tonIN
	CAL	timer_7
after_start_timer_7:
	JMP	end
	(* The conditions *)
check_e_0:
	(* Condition for event arm.allocate_lower_buffer *)
	LD	e_0
	JMPCN	after_check_e_0
	JMP	after_check_e_0
check_e_1:
	(* Condition for event arm.allocate_upper_buffer *)
	LD	e_1
	JMPCN	after_check_e_1
	JMP	after_check_e_1
check_e_2:
	(* Condition for event arm.lower_lower_buffer *)
	LD	e_2
	JMPCN	after_check_e_2
	JMP	after_check_e_2
check_e_3:
	(* Condition for event arm.lower_upper_buffer *)
	LD	e_3
	JMPCN	after_check_e_3
	JMP	after_check_e_3
check_e_4:
	(* Condition for event arm.raise_lower_buffer *)
	LD	e_4
	JMPCN	after_check_e_4
	JMP	after_check_e_4
check_e_5:
	(* Condition for event arm.raise_upper_buffer *)
	LD	e_5
	JMPCN	after_check_e_5
	JMP	after_check_e_5
check_e_6:
	(* Condition for event arm.release_lower_buffer *)
	LD	e_6
	JMPCN	after_check_e_6
	JMP	after_check_e_6
check_e_7:
	(* Condition for event arm.release_upper_buffer *)
	LD	e_7
	JMPCN	after_check_e_7
	JMP	after_check_e_7
check_e_8:
	(* Condition for event button.automatic.pressed *)
	LD	e_8
	JMPCN	after_check_e_8
	LD	si_23
	JMPCN	check_e_8_0
	LD	FALSE
	ST	e_8
	JMP	after_check_e_8
check_e_8_0:
	JMP	after_check_e_8
check_e_9:
	(* Condition for event button.automatic.released *)
	LD	e_9
	JMPCN	after_check_e_9
	LD	si_23
	JMPC	check_e_9_0
	LD	FALSE
	ST	e_9
	JMP	after_check_e_9
check_e_9_0:
	JMP	after_check_e_9
check_e_10:
	(* Condition for event button.manual.pressed *)
	LD	e_10
	JMPCN	after_check_e_10
	LD	si_24
	JMPCN	check_e_10_0
	LD	FALSE
	ST	e_10
	JMP	after_check_e_10
check_e_10_0:
	JMP	after_check_e_10
check_e_11:
	(* Condition for event button.manual.released *)
	LD	e_11
	JMPCN	after_check_e_11
	LD	si_24
	JMPC	check_e_11_0
	LD	FALSE
	ST	e_11
	JMP	after_check_e_11
check_e_11_0:
	JMP	after_check_e_11
check_e_12:
	(* Condition for event em.ball_out_of_measure_station *)
	LD	e_12
	JMPCN	after_check_e_12
	JMP	after_check_e_12
check_e_13:
	(* Condition for event em.elevator.allocate_station *)
	LD	e_13
	JMPCN	after_check_e_13
	JMP	after_check_e_13
check_e_14:
	(* Condition for event em.elevator.release_station *)
	LD	e_14
	JMPCN	after_check_e_14
	JMP	after_check_e_14
check_e_15:
	(* Condition for event em.enter_ball *)
	LD	e_15
	JMPCN	after_check_e_15
	JMP	after_check_e_15
check_e_16:
	(* Condition for event em.go_down *)
	LD	e_16
	JMPCN	after_check_e_16
	JMP	after_check_e_16
check_e_17:
	(* Condition for event em.go_up *)
	LD	e_17
	JMPCN	after_check_e_17
	JMP	after_check_e_17
check_e_18:
	(* Condition for event em.has_ball *)
	LD	e_18
	JMPCN	after_check_e_18
	LD	si_2
	JMPC	check_e_18_0
	LD	FALSE
	ST	e_18
	JMP	after_check_e_18
check_e_18_0:
	JMP	after_check_e_18
check_e_19:
	(* Condition for event em.is_down *)
	LD	e_19
	JMPCN	after_check_e_19
	LD	si_1
	JMPC	check_e_19_0
	LD	FALSE
	ST	e_19
	JMP	after_check_e_19
check_e_19_0:
	JMP	after_check_e_19
check_e_20:
	(* Condition for event em.is_up *)
	LD	e_20
	JMPCN	after_check_e_20
	LD	si_3
	JMPC	check_e_20_0
	LD	FALSE
	ST	e_20
	JMP	after_check_e_20
check_e_20_0:
	JMP	after_check_e_20
check_e_21:
	(* Condition for event em.large_ball *)
	LD	e_21
	JMPCN	after_check_e_21
	LD	si_5
	JMPC	check_e_21_0
	LD	FALSE
	ST	e_21
	JMP	after_check_e_21
check_e_21_0:
	JMP	after_check_e_21
check_e_22:
	(* Condition for event em.measure.allocate_station *)
	LD	e_22
	JMPCN	after_check_e_22
	JMP	after_check_e_22
check_e_23:
	(* Condition for event em.measure.finished *)
	LD	e_23
	JMPCN	after_check_e_23
	JMP	after_check_e_23
check_e_24:
	(* Condition for event em.measure.go_in *)
	LD	e_24
	JMPCN	after_check_e_24
	JMP	after_check_e_24
check_e_25:
	(* Condition for event em.measure.go_out *)
	LD	e_25
	JMPCN	after_check_e_25
	JMP	after_check_e_25
check_e_26:
	(* Condition for event em.measure.has_ball *)
	LD	e_26
	JMPCN	after_check_e_26
	LD	si_4
	JMPC	check_e_26_0
	LD	FALSE
	ST	e_26
	JMP	after_check_e_26
check_e_26_0:
	JMP	after_check_e_26
check_e_27:
	(* Condition for event em.measure.has_no_ball *)
	LD	e_27
	JMPCN	after_check_e_27
	LD	si_4
	JMPCN	check_e_27_0
	LD	FALSE
	ST	e_27
	JMP	after_check_e_27
check_e_27_0:
	JMP	after_check_e_27
check_e_28:
	(* Condition for event em.measure.release_station *)
	LD	e_28
	JMPCN	after_check_e_28
	JMP	after_check_e_28
check_e_29:
	(* Condition for event em.measure.start *)
	LD	e_29
	JMPCN	after_check_e_29
	JMP	after_check_e_29
check_e_30:
	(* Condition for event em.putter.allocate_station *)
	LD	e_30
	JMPCN	after_check_e_30
	JMP	after_check_e_30
check_e_31:
	(* Condition for event em.putter.finished *)
	LD	e_31
	JMPCN	after_check_e_31
	JMP	after_check_e_31
check_e_32:
	(* Condition for event em.putter.go_in *)
	LD	e_32
	JMPCN	after_check_e_32
	JMP	after_check_e_32
check_e_33:
	(* Condition for event em.putter.go_out *)
	LD	e_33
	JMPCN	after_check_e_33
	JMP	after_check_e_33
check_e_34:
	(* Condition for event em.putter.is_in *)
	LD	e_34
	JMPCN	after_check_e_34
	JMP	after_check_e_34
check_e_35:
	(* Condition for event em.putter.is_out *)
	LD	e_35
	JMPCN	after_check_e_35
	JMP	after_check_e_35
check_e_36:
	(* Condition for event em.putter.release_station *)
	LD	e_36
	JMPCN	after_check_e_36
	JMP	after_check_e_36
check_e_37:
	(* Condition for event em.putter.start *)
	LD	e_37
	JMPCN	after_check_e_37
	JMP	after_check_e_37
check_e_38:
	(* Condition for event em.small_ball *)
	LD	e_38
	JMPCN	after_check_e_38
	LD	si_6
	JMPC	check_e_38_0
	LD	FALSE
	ST	e_38
	JMP	after_check_e_38
check_e_38_0:
	JMP	after_check_e_38
check_e_39:
	(* Condition for event em.timer.before_ballcheck.start *)
	LD	e_39
	JMPCN	after_check_e_39
	JMP	after_check_e_39
check_e_40:
	(* Condition for event em.timer.before_ballcheck.timeout *)
	LD	e_40
	JMPCN	after_check_e_40
	JMP	after_check_e_40
check_e_41:
	(* Condition for event em.timer.before_put.start *)
	LD	e_41
	JMPCN	after_check_e_41
	JMP	after_check_e_41
check_e_42:
	(* Condition for event em.timer.before_put.timeout *)
	LD	e_42
	JMPCN	after_check_e_42
	JMP	after_check_e_42
check_e_43:
	(* Condition for event em.timer.before_up.start *)
	LD	e_43
	JMPCN	after_check_e_43
	JMP	after_check_e_43
check_e_44:
	(* Condition for event em.timer.before_up.timeout *)
	LD	e_44
	JMPCN	after_check_e_44
	JMP	after_check_e_44
check_e_45:
	(* Condition for event em.timer.measure.start *)
	LD	e_45
	JMPCN	after_check_e_45
	JMP	after_check_e_45
check_e_46:
	(* Condition for event em.timer.measure.timeout *)
	LD	e_46
	JMPCN	after_check_e_46
	JMP	after_check_e_46
check_e_47:
	(* Condition for event em.timer.putting.start *)
	LD	e_47
	JMPCN	after_check_e_47
	JMP	after_check_e_47
check_e_48:
	(* Condition for event em.timer.putting.timeout *)
	LD	e_48
	JMPCN	after_check_e_48
	JMP	after_check_e_48
check_e_49:
	(* Condition for event es.allocate_lower_buffer *)
	LD	e_49
	JMPCN	after_check_e_49
	JMP	after_check_e_49
check_e_50:
	(* Condition for event es.allocate_upper_buffer *)
	LD	e_50
	JMPCN	after_check_e_50
	JMP	after_check_e_50
check_e_51:
	(* Condition for event es.ball_lower_level *)
	LD	e_51
	JMPCN	after_check_e_51
	LD	si_12
	JMPC	check_e_51_0
	LD	FALSE
	ST	e_51
	JMP	after_check_e_51
check_e_51_0:
	JMP	after_check_e_51
check_e_52:
	(* Condition for event es.ball_upper_level *)
	LD	e_52
	JMPCN	after_check_e_52
	LD	si_15
	JMPC	check_e_52_0
	LD	FALSE
	ST	e_52
	JMP	after_check_e_52
check_e_52_0:
	JMP	after_check_e_52
check_e_53:
	(* Condition for event es.deput_ball_lower *)
	LD	e_53
	JMPCN	after_check_e_53
	JMP	after_check_e_53
check_e_54:
	(* Condition for event es.deput_ball_upper *)
	LD	e_54
	JMPCN	after_check_e_54
	JMP	after_check_e_54
check_e_55:
	(* Condition for event es.enter_ball *)
	LD	e_55
	JMPCN	after_check_e_55
	JMP	after_check_e_55
check_e_56:
	(* Condition for event es.go_down *)
	LD	e_56
	JMPCN	after_check_e_56
	JMP	after_check_e_56
check_e_57:
	(* Condition for event es.got_ball *)
	LD	e_57
	JMPCN	after_check_e_57
	LD	si_10
	JMPC	check_e_57_0
	LD	FALSE
	ST	e_57
	JMP	after_check_e_57
check_e_57_0:
	JMP	after_check_e_57
check_e_58:
	(* Condition for event es.is_lower *)
	LD	e_58
	JMPCN	after_check_e_58
	LD	si_11
	JMPC	check_e_58_0
	LD	FALSE
	ST	e_58
	JMP	after_check_e_58
check_e_58_0:
	JMP	after_check_e_58
check_e_59:
	(* Condition for event es.is_not_down *)
	LD	e_59
	JMPCN	after_check_e_59
	JMP	after_check_e_59
check_e_60:
	(* Condition for event es.is_upper *)
	LD	e_60
	JMPCN	after_check_e_60
	LD	si_14
	JMPC	check_e_60_0
	LD	FALSE
	ST	e_60
	JMP	after_check_e_60
check_e_60_0:
	JMP	after_check_e_60
check_e_61:
	(* Condition for event es.lower_putter.go_in *)
	LD	e_61
	JMPCN	after_check_e_61
	JMP	after_check_e_61
check_e_62:
	(* Condition for event es.lower_putter.go_out *)
	LD	e_62
	JMPCN	after_check_e_62
	JMP	after_check_e_62
check_e_63:
	(* Condition for event es.no_ball_lower_level *)
	LD	e_63
	JMPCN	after_check_e_63
	LD	si_12
	JMPCN	check_e_63_0
	LD	FALSE
	ST	e_63
	JMP	after_check_e_63
check_e_63_0:
	JMP	after_check_e_63
check_e_64:
	(* Condition for event es.no_ball_upper_level *)
	LD	e_64
	JMPCN	after_check_e_64
	LD	si_15
	JMPCN	check_e_64_0
	LD	FALSE
	ST	e_64
	JMP	after_check_e_64
check_e_64_0:
	JMP	after_check_e_64
check_e_65:
	(* Condition for event es.put_ball_lower *)
	LD	e_65
	JMPCN	after_check_e_65
	JMP	after_check_e_65
check_e_66:
	(* Condition for event es.put_ball_upper *)
	LD	e_66
	JMPCN	after_check_e_66
	JMP	after_check_e_66
check_e_67:
	(* Condition for event es.release_lower_buffer *)
	LD	e_67
	JMPCN	after_check_e_67
	JMP	after_check_e_67
check_e_68:
	(* Condition for event es.release_upper_buffer *)
	LD	e_68
	JMPCN	after_check_e_68
	JMP	after_check_e_68
check_e_69:
	(* Condition for event es.timer.before_ballcheck.start *)
	LD	e_69
	JMPCN	after_check_e_69
	JMP	after_check_e_69
check_e_70:
	(* Condition for event es.timer.before_ballcheck.timeout *)
	LD	e_70
	JMPCN	after_check_e_70
	JMP	after_check_e_70
check_e_71:
	(* Condition for event es.timer.before_deput.start *)
	LD	e_71
	JMPCN	after_check_e_71
	JMP	after_check_e_71
check_e_72:
	(* Condition for event es.timer.before_deput.timeout *)
	LD	e_72
	JMPCN	after_check_e_72
	JMP	after_check_e_72
check_e_73:
	(* Condition for event es.timer.before_up.start *)
	LD	e_73
	JMPCN	after_check_e_73
	JMP	after_check_e_73
check_e_74:
	(* Condition for event es.timer.before_up.timeout *)
	LD	e_74
	JMPCN	after_check_e_74
	JMP	after_check_e_74
check_e_75:
	(* Condition for event es.up_lower *)
	LD	e_75
	JMPCN	after_check_e_75
	JMP	after_check_e_75
check_e_76:
	(* Condition for event es.up_upper *)
	LD	e_76
	JMPCN	after_check_e_76
	JMP	after_check_e_76
check_e_77:
	(* Condition for event es.upper_putter.go_in *)
	LD	e_77
	JMPCN	after_check_e_77
	JMP	after_check_e_77
check_e_78:
	(* Condition for event es.upper_putter.go_out *)
	LD	e_78
	JMPCN	after_check_e_78
	JMP	after_check_e_78
check_e_79:
	(* Condition for event gk.ball_out_of_gatekeeper *)
	LD	e_79
	JMPCN	after_check_e_79
	JMP	after_check_e_79
check_e_80:
	(* Condition for event gk.enter_ball *)
	LD	e_80
	JMPCN	after_check_e_80
	JMP	after_check_e_80
check_e_81:
	(* Condition for event gk.has_ball *)
	LD	e_81
	JMPCN	after_check_e_81
	LD	si_0
	JMPC	check_e_81_0
	LD	FALSE
	ST	e_81
	JMP	after_check_e_81
check_e_81_0:
	JMP	after_check_e_81
check_e_82:
	(* Condition for event gk.in.go_in *)
	LD	e_82
	JMPCN	after_check_e_82
	JMP	after_check_e_82
check_e_83:
	(* Condition for event gk.in.go_out *)
	LD	e_83
	JMPCN	after_check_e_83
	JMP	after_check_e_83
check_e_84:
	(* Condition for event gk.in.is_in *)
	LD	e_84
	JMPCN	after_check_e_84
	JMP	after_check_e_84
check_e_85:
	(* Condition for event gk.in.is_out *)
	LD	e_85
	JMPCN	after_check_e_85
	JMP	after_check_e_85
check_e_86:
	(* Condition for event gk.out.go_in *)
	LD	e_86
	JMPCN	after_check_e_86
	JMP	after_check_e_86
check_e_87:
	(* Condition for event gk.out.go_out *)
	LD	e_87
	JMPCN	after_check_e_87
	JMP	after_check_e_87
check_e_88:
	(* Condition for event gk.out.is_in *)
	LD	e_88
	JMPCN	after_check_e_88
	JMP	after_check_e_88
check_e_89:
	(* Condition for event gk.out.is_out *)
	LD	e_89
	JMPCN	after_check_e_89
	JMP	after_check_e_89
check_e_90:
	(* Condition for event gk.release_ball *)
	LD	e_90
	JMPCN	after_check_e_90
	JMP	after_check_e_90
check_e_91:
	(* Condition for event is_large_ball *)
	LD	e_91
	JMPCN	after_check_e_91
	JMP	after_check_e_91
check_e_92:
	(* Condition for event is_small_ball *)
	LD	e_92
	JMPCN	after_check_e_92
	JMP	after_check_e_92
check_e_93:
	(* Condition for event mode.automatic *)
	LD	e_93
	JMPCN	after_check_e_93
	JMP	after_check_e_93
check_e_94:
	(* Condition for event mode.manual *)
	LD	e_94
	JMPCN	after_check_e_94
	JMP	after_check_e_94
	(* The actions *)
do_e_0:
	(* Action for event arm.allocate_lower_buffer *)
	JMP	after_do_e_0
do_e_1:
	(* Action for event arm.allocate_upper_buffer *)
	JMP	after_do_e_1
do_e_2:
	(* Action for event arm.lower_lower_buffer *)
	JMP	after_do_e_2
do_e_3:
	(* Action for event arm.lower_upper_buffer *)
	JMP	after_do_e_3
do_e_4:
	(* Action for event arm.raise_lower_buffer *)
	JMP	after_do_e_4
do_e_5:
	(* Action for event arm.raise_upper_buffer *)
	JMP	after_do_e_5
do_e_6:
	(* Action for event arm.release_lower_buffer *)
	JMP	after_do_e_6
do_e_7:
	(* Action for event arm.release_upper_buffer *)
	JMP	after_do_e_7
do_e_8:
	(* Action for event button.automatic.pressed *)
	JMP	after_do_e_8
do_e_9:
	(* Action for event button.automatic.released *)
	JMP	after_do_e_9
do_e_10:
	(* Action for event button.manual.pressed *)
	JMP	after_do_e_10
do_e_11:
	(* Action for event button.manual.released *)
	JMP	after_do_e_11
do_e_12:
	(* Action for event em.ball_out_of_measure_station *)
	JMP	after_do_e_12
do_e_13:
	(* Action for event em.elevator.allocate_station *)
	JMP	after_do_e_13
do_e_14:
	(* Action for event em.elevator.release_station *)
	JMP	after_do_e_14
do_e_15:
	(* Action for event em.enter_ball *)
	JMP	after_do_e_15
do_e_16:
	(* Action for event em.go_down *)
	LD	FALSE
	ST	so_2
	JMP	after_do_e_16
do_e_17:
	(* Action for event em.go_up *)
	LD	TRUE
	ST	so_2
	JMP	after_do_e_17
do_e_18:
	(* Action for event em.has_ball *)
	JMP	after_do_e_18
do_e_19:
	(* Action for event em.is_down *)
	JMP	after_do_e_19
do_e_20:
	(* Action for event em.is_up *)
	JMP	after_do_e_20
do_e_21:
	(* Action for event em.large_ball *)
	JMP	after_do_e_21
do_e_22:
	(* Action for event em.measure.allocate_station *)
	JMP	after_do_e_22
do_e_23:
	(* Action for event em.measure.finished *)
	JMP	after_do_e_23
do_e_24:
	(* Action for event em.measure.go_in *)
	LD	FALSE
	ST	so_4
	JMP	after_do_e_24
do_e_25:
	(* Action for event em.measure.go_out *)
	LD	TRUE
	ST	so_4
	JMP	after_do_e_25
do_e_26:
	(* Action for event em.measure.has_ball *)
	JMP	after_do_e_26
do_e_27:
	(* Action for event em.measure.has_no_ball *)
	JMP	after_do_e_27
do_e_28:
	(* Action for event em.measure.release_station *)
	JMP	after_do_e_28
do_e_29:
	(* Action for event em.measure.start *)
	JMP	after_do_e_29
do_e_30:
	(* Action for event em.putter.allocate_station *)
	JMP	after_do_e_30
do_e_31:
	(* Action for event em.putter.finished *)
	JMP	after_do_e_31
do_e_32:
	(* Action for event em.putter.go_in *)
	LD	FALSE
	ST	so_3
	JMP	after_do_e_32
do_e_33:
	(* Action for event em.putter.go_out *)
	LD	TRUE
	ST	so_3
	JMP	after_do_e_33
do_e_34:
	(* Action for event em.putter.is_in *)
	JMP	after_do_e_34
do_e_35:
	(* Action for event em.putter.is_out *)
	JMP	after_do_e_35
do_e_36:
	(* Action for event em.putter.release_station *)
	JMP	after_do_e_36
do_e_37:
	(* Action for event em.putter.start *)
	JMP	after_do_e_37
do_e_38:
	(* Action for event em.small_ball *)
	JMP	after_do_e_38
do_e_39:
	(* Action for event em.timer.before_ballcheck.start *)
	JMP	after_do_e_39
do_e_40:
	(* Action for event em.timer.before_ballcheck.timeout *)
	JMP	after_do_e_40
do_e_41:
	(* Action for event em.timer.before_put.start *)
	JMP	after_do_e_41
do_e_42:
	(* Action for event em.timer.before_put.timeout *)
	JMP	after_do_e_42
do_e_43:
	(* Action for event em.timer.before_up.start *)
	JMP	after_do_e_43
do_e_44:
	(* Action for event em.timer.before_up.timeout *)
	JMP	after_do_e_44
do_e_45:
	(* Action for event em.timer.measure.start *)
	JMP	after_do_e_45
do_e_46:
	(* Action for event em.timer.measure.timeout *)
	JMP	after_do_e_46
do_e_47:
	(* Action for event em.timer.putting.start *)
	JMP	after_do_e_47
do_e_48:
	(* Action for event em.timer.putting.timeout *)
	JMP	after_do_e_48
do_e_49:
	(* Action for event es.allocate_lower_buffer *)
	JMP	after_do_e_49
do_e_50:
	(* Action for event es.allocate_upper_buffer *)
	JMP	after_do_e_50
do_e_51:
	(* Action for event es.ball_lower_level *)
	JMP	after_do_e_51
do_e_52:
	(* Action for event es.ball_upper_level *)
	JMP	after_do_e_52
do_e_53:
	(* Action for event es.deput_ball_lower *)
	JMP	after_do_e_53
do_e_54:
	(* Action for event es.deput_ball_upper *)
	JMP	after_do_e_54
do_e_55:
	(* Action for event es.enter_ball *)
	JMP	after_do_e_55
do_e_56:
	(* Action for event es.go_down *)
	LD	FALSE
	ST	so_5
	LD	FALSE
	ST	so_6
	JMP	after_do_e_56
do_e_57:
	(* Action for event es.got_ball *)
	JMP	after_do_e_57
do_e_58:
	(* Action for event es.is_lower *)
	JMP	after_do_e_58
do_e_59:
	(* Action for event es.is_not_down *)
	JMP	after_do_e_59
do_e_60:
	(* Action for event es.is_upper *)
	JMP	after_do_e_60
do_e_61:
	(* Action for event es.lower_putter.go_in *)
	LD	FALSE
	ST	so_7
	JMP	after_do_e_61
do_e_62:
	(* Action for event es.lower_putter.go_out *)
	LD	TRUE
	ST	so_7
	JMP	after_do_e_62
do_e_63:
	(* Action for event es.no_ball_lower_level *)
	JMP	after_do_e_63
do_e_64:
	(* Action for event es.no_ball_upper_level *)
	JMP	after_do_e_64
do_e_65:
	(* Action for event es.put_ball_lower *)
	JMP	after_do_e_65
do_e_66:
	(* Action for event es.put_ball_upper *)
	JMP	after_do_e_66
do_e_67:
	(* Action for event es.release_lower_buffer *)
	JMP	after_do_e_67
do_e_68:
	(* Action for event es.release_upper_buffer *)
	JMP	after_do_e_68
do_e_69:
	(* Action for event es.timer.before_ballcheck.start *)
	JMP	after_do_e_69
do_e_70:
	(* Action for event es.timer.before_ballcheck.timeout *)
	JMP	after_do_e_70
do_e_71:
	(* Action for event es.timer.before_deput.start *)
	JMP	after_do_e_71
do_e_72:
	(* Action for event es.timer.before_deput.timeout *)
	JMP	after_do_e_72
do_e_73:
	(* Action for event es.timer.before_up.start *)
	JMP	after_do_e_73
do_e_74:
	(* Action for event es.timer.before_up.timeout *)
	JMP	after_do_e_74
do_e_75:
	(* Action for event es.up_lower *)
	LD	TRUE
	ST	so_5
	LD	FALSE
	ST	so_6
	JMP	after_do_e_75
do_e_76:
	(* Action for event es.up_upper *)
	LD	TRUE
	ST	so_5
	LD	TRUE
	ST	so_6
	JMP	after_do_e_76
do_e_77:
	(* Action for event es.upper_putter.go_in *)
	LD	FALSE
	ST	so_11
	JMP	after_do_e_77
do_e_78:
	(* Action for event es.upper_putter.go_out *)
	LD	TRUE
	ST	so_11
	JMP	after_do_e_78
do_e_79:
	(* Action for event gk.ball_out_of_gatekeeper *)
	JMP	after_do_e_79
do_e_80:
	(* Action for event gk.enter_ball *)
	JMP	after_do_e_80
do_e_81:
	(* Action for event gk.has_ball *)
	JMP	after_do_e_81
do_e_82:
	(* Action for event gk.in.go_in *)
	LD	FALSE
	ST	so_0
	JMP	after_do_e_82
do_e_83:
	(* Action for event gk.in.go_out *)
	LD	TRUE
	ST	so_0
	JMP	after_do_e_83
do_e_84:
	(* Action for event gk.in.is_in *)
	JMP	after_do_e_84
do_e_85:
	(* Action for event gk.in.is_out *)
	JMP	after_do_e_85
do_e_86:
	(* Action for event gk.out.go_in *)
	LD	FALSE
	ST	so_1
	JMP	after_do_e_86
do_e_87:
	(* Action for event gk.out.go_out *)
	LD	TRUE
	ST	so_1
	JMP	after_do_e_87
do_e_88:
	(* Action for event gk.out.is_in *)
	JMP	after_do_e_88
do_e_89:
	(* Action for event gk.out.is_out *)
	JMP	after_do_e_89
do_e_90:
	(* Action for event gk.release_ball *)
	JMP	after_do_e_90
do_e_91:
	(* Action for event is_large_ball *)
	JMP	after_do_e_91
do_e_92:
	(* Action for event is_small_ball *)
	JMP	after_do_e_92
do_e_93:
	(* Action for event mode.automatic *)
	JMP	after_do_e_93
do_e_94:
	(* Action for event mode.manual *)
	JMP	after_do_e_94
end:
END_PROGRAM
(* JAVA_BLOCKS for printing (no newline) *)
(*=======================================*)
